(* IEC 61131-3 sources: ConveyorControl-with-PLC/4E_Gruppe1_Graf_Projekt1_HMI/Class/_Lse (part 2) *)

StrChrUniBbB
    LDRB      r3, [p0], #1
    LDRB      r11, [p0], #1
    ORR       r3, r3, r11, LSL #8
    CMP       r3, x1
    BEQ       StrChrEnd
    CMP       r3, #0
    BEQ       StrChrNotFound
    ADD       r10, r10, #1
    B         StrChrUniBbB

StrChrNotFound
    MOV       r10, #65280
    ADD       r10, r10, #255

StrChrEnd
    MOV       retcode, r10
#else //elif _LSL_TARGETARCH_X86
    pushfd
    push      esi

    clr       ebx
    clr       ecx

    l.esi     p0
    o.esi     esi
    jz        StringChrRet

    cld
    l.bx      x1
    cmp.w     x2,1
    jne       StringChrLoopUni

StringChrLoop
    lodsb
    o.al      al
    jz        StringChrRet
    x.al      bl
    jz        StringChrSuccess
    inc       ecx
    jmp       StringChrLoop

StringChrLoopUni
    lodsw
    o.ax      ax
    jz        StringChrRet
    x.ax      bx
    jz        StringChrSuccess
    inc       ecx
    jmp       StringChrLoopUni

StringChrRet
    l.ecx     16#FFFF

StringChrSuccess
    s.cx      retcode

    pop       esi
    popfd
#endif

END_FUNCTION

FUNCTION AWL GLOBAL __CDECL StrXmp
  VAR_INPUT
    pTxt0    : ^void;
    pTxt1    : ^void;
    cSize : UINT;
  END_VAR
  VAR_OUTPUT
    retcode : UDINT;
  END_VAR

#ifdef _LSL_TARGETARCH_ARM
    MOV       retcode, #0

    CMP       pTxt0, pTxt1
    BEQ       StrXmpEnd

    CMP       pTxt0, #0
    BEQ       StrXmpNotEqual
    CMP       pTxt1, #0
    BEQ       StrXmpNotEqual

    CMP       cSize, #1
    BNE       StrXmpUni

StrXmpAscii
    LDRB      r10, [pTxt0], #1
    LDRB      r11, [pTxt1], #1
    CMP       r10, r11
    BNE       StrXmpNotEqual
    CMP       r10, #0
    BEQ       StrXmpEnd
    B         StrXmpAscii

StrXmpUni
    ORR       r11, pTxt0, pTxt1
    TST       r11, #1
    BNE       StrXmpUniBbB   // one or both pointer are missaligned

StrXmpUniH
    LDRH      r10, [pTxt0], #2
    LDRH      r11, [pTxt1], #2
    CMP       r10, r11
    BNE       StrXmpNotEqual
    CMP       r10, #0
    BNE       StrXmpUniH
    B         StrXmpEnd

StrXmpUniBbB
    LDRB      r10, [pTxt0], #1
    LDRB      r3,  [pTxt0], #1
    ORR       r10, r10, r3, LSL #8
    LDRB      r11, [pTxt1], #1
    LDRB      r3,  [pTxt1], #1
    ORR       r11, r11, r3, LSL #8
    CMP       r10, r11
    BNE       StrXmpNotEqual
    CMP       r10, #0
    BNE       StrXmpUniBbB
    B         StrXmpEnd

StrXmpNotEqual
    MOV       retcode, #1

StrXmpEnd

#else //elif _LSL_TARGETARCH_X86
    pushfd
    push      edi
    push      esi

    l.esi     pTxt0
    l.edi     pTxt1
    clr       ecx

    x.esi     edi
    jz        StringXmpEqual

    l.esi     pTxt0
    o.esi     esi
    jz        StringXmpRet
    o.edi     edi
    jz        StringXmpRet

    cld
    cmp.w     cSize,1
    jne       StringXmpLoopUni

StringXmpLoop
    l.cl      (edi)
    or.cl     (esi)
    jecxz     StringXmpEqual
    cmpsb
    jz        StringXmpLoop
    jmp       StringXmpRet

StringXmpLoopUni
    l.cx      (edi)
    or.cx     (esi)
    jecxz     StringXmpEqual
    cmpsw
    jz        StringXmpLoopUni
    //jmp       StringXmpRet

StringXmpRet
    l.ecx     1

StringXmpEqual
    s.ecx     retcode

    pop       esi
    pop       edi

    popfd
#endif

END_FUNCTION

FUNCTION GLOBAL __CDECL get_loaderversion
VAR_OUTPUT
  retcode : UDINT;
END_VAR

  retcode := ops.uiLoaderVersion.usLoRev or (ops.uiLoaderVersion.usHiRev shl 16);

END_FUNCTION

FUNCTION _LookupCls VAR_INPUT pname : ^char; END_VAR VAR_OUTPUT retcode : ^CLSHDR; END_VAR;
FUNCTION GLOBAL __cdecl GetRevisionOfClass VAR_INPUT classname : ^char; END_VAR VAR_OUTPUT retcode : udint; END_VAR
  var
    pClsHdr : ^CLSHDR;
    rhi, rlo : udint;
  end_var

  retcode := 0;
  pClsHdr := _LookupCls(classname);

  if(pClsHdr <> NIL) then
    if(pClsHdr^.pDsc <> NIL) then
      rhi := pClsHdr^.pDsc^.udRev.hi;
      rlo := pClsHdr^.pDsc^.udRev.lo;
      retcode := (rhi shl 16) or rlo;
    end_if;
  end_if;

END_FUNCTION

FUNCTION GLOBAL __CDECL rotate_DOT
VAR_INPUT
  p    : ^_DOT;
  w1   : INT;
END_VAR
VAR
  a1, x, y : _REAL;
  m0, m1 : _REAL;
END_VAR

  x := p^.x;
  y := p^.y;

  a1 := (to_real(w1) * 3.1416) / 180;
  m0 := COS(a1);
  m1 := SIN(a1);

  p^.x := to_int((m0 * x) + (m1 * y));
  p^.y := to_int((m0 * y) - (m1 * x));

END_FUNCTION

FUNCTION GLOBAL __CDECL matrize
VAR_INPUT
  pm : ^_REAL;
  px : ^_REAL;
  py : ^_REAL;
  pz : ^_REAL;
END_VAR
VAR
  x : _REAL;
  y : _REAL;
  z : _REAL;
END_VAR

  x := px^;
  y := py^;
  z := pz^;

  px^ :=( pm^ * x) + ((pm + sizeof(_REAL))^ * y) + ((pm + (sizeof(_REAL) * 2))^ * z);
  py^ := ((pm + (sizeof(_REAL) * 3))^ * x) + ((pm + (sizeof(_REAL) * 4))^ * y) + ((pm + (sizeof(_REAL) * 5))^ * z);
  pz^ := ((pm + (sizeof(_REAL) * 6))^ * x) + ((pm + (sizeof(_REAL) * 7))^ * y) + ((pm + (sizeof(_REAL) * 8))^ * z);

END_FUNCTION

FUNCTION GLOBAL __CDECL rotate_DOT3D
VAR_INPUT
  p    : ^_DOT3D;
  w1   : INT;
  w2   : INT;
  w3   : INT;
END_VAR
VAR
  a1   : _REAL;
  a2   : _REAL;
  a3   : _REAL;
  x    : _REAL;
  y    : _REAL;
  z    : _REAL;
  matr : ARRAY[0..8] of _REAL;
END_VAR

  a1 := w1;
  a2 := w2;
  a3 := w3;

  a1 := (a1 * 3.1416) / 180;
  a2 := (a2 * 3.1416) / 180;
  a3 := (a3 * 3.1416) / 180;

  x := p^.x;
  y := p^.y;
  z := p^.z;

  matr[0] := COS(a1);
  matr[1] := SIN(a1);
  matr[2] := 0;
  matr[3] := -matr[1];
  matr[4] := matr[0];
  matr[5] := 0;
  matr[6] := 0;
  matr[7] := 0;
  matr[8] := 1;
  matrize(#matr[0], #x, #y, #z);

  matr[0] := 1;
  matr[1] := 0;
  matr[2] := 0;
  matr[3] := 0;
  matr[4] := COS(a2);
  matr[5] := SIN(a2);
  matr[6] := 0;
  matr[7] := -matr[5];
  matr[8] := matr[4];
  matrize(#matr[0], #x, #y, #z);

  matr[0] := COS(a3);
  matr[1] := 0;
  matr[2] := SIN(a3);
  matr[3] := 0;
  matr[4] := 1;
  matr[5] := 0;
  matr[6] := -matr[2];
  matr[7] := 0;
  matr[8] := matr[0];
  matrize(#matr[0], #x, #y, #z);

//  p^.x := FTOL(x);
//  p^.y := FTOL(y);
//  p^.z := FTOL(z);

  p^.x := to_int(x);
  p^.y := to_int(y);
  p^.z := to_int(z);

END_FUNCTION

FUNCTION GLOBAL __CDECL AMBDC
VAR_INPUT
  a : UDINT;
  b : UDINT;
  c : UDINT;
END_VAR
VAR_OUTPUT
  retcode : UDINT;
END_VAR

  retcode := a*b/c;

END_FUNCTION

FUNCTION GLOBAL __CDECL heap_size
VAR_INPUT
  total : ^UDINT;
  free  : ^UDINT;
END_VAR
VAR_OUTPUT
  retcode : bool;
END_VAR

  free^  := _UserHeapFreeMem;
  total^ := _UserHeapTotalSize;
  retcode := true;

END_FUNCTION

FUNCTION GLOBAL __CDECL get_microtime
VAR_OUTPUT
  retcode : UDINT;
END_VAR

  retcode := OS_ReadMicroSec();

END_FUNCTION

FUNCTION GLOBAL __CDECL GetResetTaskTime
VAR_INPUT
  pudi : ^UDINT;
END_VAR

  if(pudi <> NIL) then
    pudi^ := _RealMaximumTime;       pudi += 4; // maximum duration of RT-methods
    pudi^ := _RealAverageTime;       pudi += 4; // average duration of RT-methods
    pudi^ := _CyclicMaximumTime;     pudi += 4; // maximum duration of Cy-methods
    pudi^ := _CyclicAverageTime;     pudi += 4; // average duration of Cy-methods
    pudi^ := _BackgroundMaximumTime; pudi += 4; // maximum duration of Bg-methods
    pudi^ := _BackgroundAverageTime;            // average duration of Bg-methods
  else
    _RealMaximumTime       := 0;  // maximum duration of RT-methods
    _RealAverageTime       := 0;  // average duration of RT-methods
    _CyclicMaximumTime     := 0;  // maximum duration of Cy-methods
    _CyclicAverageTime     := 0;  // average duration of Cy-methods
    _BackgroundMaximumTime := 0;  // maximum duration of Bg-methods
    _BackgroundAverageTime := 0;  // average duration of Bg-methods
  end_if;

END_FUNCTION

FUNCTION GLOBAL __CDECL CilGet
VAR_INPUT
	name : ^_ASCII;
	ptr  : ^PVOID;
END_VAR
VAR_OUTPUT
	retcode : BOOL;
END_VAR

  retcode := TRUE;

  if(OS_CILGet(name, ptr) <> SYS_ERR_NONE) then
    ptr^    := NIL;
	retcode := FALSE;
  end_if;

END_FUNCTION

FUNCTION GLOBAL __CDECL GetTCPIPAddressFromDNS
VAR_INPUT
  dnsname   : ^_ASCII;
END_VAR
VAR_OUTPUT
  retcode : UDINT;
END_VAR

  retcode := 0;
  if((lsl_tcp_user <> NIL) & (dnsname <> NIL)) then
    retcode := OS_TCP_USER_STRTOULONG(dnsname);
  end_if;

END_FUNCTION

FUNCTION GLOBAL __CDECL GetTCPIPAddress
VAR_INPUT
  interface : UDINT;
  address   : ^UDINT;
  subnet    : ^UDINT;
  gateway   : ^UDINT;
END_VAR
VAR_OUTPUT
  retcode : BOOL;
END_VAR

  retcode := FALSE;

  if(lsl_tcp_user <> NIL) then
    if(address <> NIL) then
      address^ := 0;
      OS_TCP_USER_IPINFO(interface$DINT, IP_OPT_ADDR, address);
      retcode := TRUE;
    end_if;
    if(subnet <> NIL) then
      subnet^ := 0;
      OS_TCP_USER_IPINFO(interface$DINT, IP_OPT_SUBNETMASK, subnet);
      retcode := TRUE;
    end_if;
    if(gateway <> NIL) then
      gateway^ := 0;
      OS_TCP_USER_IPINFO(interface$DINT, IP_OPT_GATEWAY, gateway);
      retcode := TRUE;
    end_if;
  end_if;

END_FUNCTION

FUNCTION  _Lse::_Lse
VAR_OUTPUT
	ret_code		: CONFSTATES;
END_VAR
VAR
  i : UINT;
  ptr : ^_PICPOI;
END_VAR

  PThis_Lse      := this;
  DownloadState  := 0;
  GlobalBitState := 0;
//LDR_SetWait4Visu(true, 0);

  construct_MAIN();

  mt_api         := NIL;
  Thread2Handle  := NIL;
  MailBox2Handle := NIL;

  if(OS_CILGet("LSL_MULTITASK", #mt_api$void)) THEN
    mt_api := NIL;
  end_if;

  MutexHandler[0] := OS_MT_CreateSemaphore(MTSEMATYPE_MUTEX, 1, 0, "KERNELMUTEX");
  MutexHandler[1] := OS_MT_CreateSemaphore(MTSEMATYPE_MUTEX, 1, 0, "ALARMMUTEX");
  MutexHandler[2] := OS_MT_CreateSemaphore(MTSEMATYPE_MUTEX, 1, 0, "RTK2TASK");
  MutexHandler[3] := OS_MT_CreateSemaphore(MTSEMATYPE_MUTEX, 1, 0, "ReallocREFLIST");
  MutexHandler[4] := OS_MT_CreateSemaphore(MTSEMATYPE_MUTEX, 1, 0, "StartREFLIST");

  OS_pLslSysMsg := NIL;
  if(OS_CILGet("SYSMSG", #OS_pLslSysMsg$void)) THEN
    OS_pLslSysMsg := NIL;
  end_if;

  lsl_tcp_user := NIL;
  if(OS_CILGet("TCP_USER", #lsl_tcp_user$void)) then
    lsl_tcp_user := NIL;
  end_if;

//  init_MAIN();
  init_MEM_POINTERPARA(#UserGlobal);
  init_MEM_POINTER(#Oszis);

  ToolCat    := NIL;
  RunState   := STATE_START;
  ret_code   := C_OK;
  PicMemo.no := 0;
  ptr        := #PicMemo.ptr[0];
  i          := sizeof(PicMemo.ptr) / sizeof(_PICPOI);
  while(i) do
    init_WHOAMI(#ptr^.whoami);
	  ptr^.ptr := NIL;
	  ptr      += sizeof(_PICPOI);
    i        -= 1;
  end_while;

  IsEventProcessor := FALSE;

END_FUNCTION

FUNCTION VIRTUAL GLOBAL _Lse::Init
var
  urinit : bool;
end_var

  if((RunState = STATE_START) | (RunState = STATE_FLY)) then
    urinit := true;
	  if(RunState = STATE_FLY) then
	    urinit := false;
	  end_if;
    RunState := STATE_READY;

    if(RTK_Init(this, urinit) = FALSE) then
	    RunState := STATE_END;
    end_if;
  end_if;

  if(_firstscan) then
    if(IsClientConnected(#EventProcessor) = TRUE) then
      IsEventProcessor := TRUE;
    end_if;

    InitJpgLib();

    if(mt_api <> NIL) then
      if(MailBox2Handle = NIL) then
        MailBox2Handle := OS_MT_CreateMailBox(sizeof(_Thread2CmdLine), 16, "MyMailBox2");
      end_if;

      if(MailBox2Handle <> NIL) & (Thread2Handle = NIL) then
        Thread2Handle := OS_MT_CreateThread(#Thread2(), 9, 8192, 0, this, "MyThread2");
      end_if;
    end_if;
  end_if;

END_FUNCTION

FUNCTION VIRTUAL GLOBAL _Lse::CyWork
VAR_INPUT
EAX		: UDINT;
END_VAR
VAR_OUTPUT
	state		: UDINT;
END_VAR

  state := Background(0);

END_FUNCTION

FUNCTION VIRTUAL GLOBAL _Lse::Background
VAR_INPUT
 EAX  : UDINT;
END_VAR
VAR_OUTPUT
 state  : UDINT;
END_VAR

  if((ops.sysstate = C_RUNRAM) | (ops.sysstate = C_RUNROM)) then

    if(DownloadState = 2) then
      DownloadState := 0;
      new_PLC();
      RTK_End(TRUE);
      RunState := STATE_FLY;
      OfflineMode := 0;
      Init();
    end_if;

    if(RunState = STATE_RUN) then
      if(RTK_Run() = FALSE) then
        if(IF_Stop() = TRUE) then
          MakeLogfile1Entry("End of LSE-task forced by program.", 0, 0);
          RunState := STATE_END;
        end_if;
      end_if;
    elsif(RunState = STATE_READY) then
      RunState   := STATE_RUN;
      if(RTK_Ready() = FALSE) then
        RunState := STATE_END;
      end_if;
    elsif(RunState = STATE_END) then
      RTK_End(FALSE);
      RunState := STATE_ERROR;
    end_if;
  end_if;

  state := READY$UDINT;

END_FUNCTION

FUNCTION __CDECL VIRTUAL GLOBAL _Lse::IF_WindowStart
VAR_INPUT
	whoami		: ^_WHOAMI;
	pic		    : ^VOID;
	firsttime	: BOOL;
END_VAR
VAR
  pp  : ^_PICPOI;
	no  : UDINT;
  ppp : ^_POINTERPARA;
END_VAR

  if(GlobalBitState and GLOBAL_BIT_IFWINSTART) then
    no  := UserGlobal.no;
    ppp := UserGlobal.ptr;
    while no do
      if(ppp^.para and GLOBAL_BIT_IFWINSTART) then
        ppp^.ptr$^_Global^.IF_WindowStart(whoami, pic, firsttime);
      end_if;
	    no  -= 1;
	    ppp += sizeof(_POINTERPARA);
    end_while;
  end_if;

  pp := FindScreen(whoami);
  if(pp <> NIL) then
    pp^.ptr$^_Screen^.S_Start(pic, firsttime);
    pic^$^_Screen := pp^.ptr$^_Screen;
  end_if;

END_FUNCTION

FUNCTION __CDECL VIRTUAL GLOBAL _Lse::IF_WindowReady
VAR_INPUT
	whoami		: ^_WHOAMI;
	pic		    : ^VOID;
	firsttime	: BOOL;
END_VAR
VAR
	no  : UDINT;
	ppp : ^_POINTERPARA;
END_VAR

  if(GlobalBitState and GLOBAL_BIT_IFWINREADY) then
    no  := UserGlobal.no;
    ppp := UserGlobal.ptr;
    while no do
      if(ppp^.para and GLOBAL_BIT_IFWINREADY) then
        ppp^.ptr$^_Global^.IF_WindowReady(whoami, pic, firsttime);
      end_if;
      no  -= 1;
      ppp += sizeof(_POINTERPARA);
    end_while;
  end_if;

  if(pic <> NIL) then
    if(pic^$^_Screen <> NIL) then
      pic^$^_Screen^.S_Ready(pic, firsttime);
    end_if;
  end_if;

END_FUNCTION

FUNCTION __CDECL VIRTUAL GLOBAL _Lse::IF_WindowRun
VAR_INPUT
	whoami		: ^_WHOAMI;
	pic		    : ^VOID;
	event		: ^_EVENT;
END_VAR
VAR
 	no  : UDINT;
	ppp : ^_POINTERPARA;
END_VAR

  if(GlobalBitState and GLOBAL_BIT_IFWINRUN) then
    no  := UserGlobal.no;
    ppp := UserGlobal.ptr;
    while no do
      if(ppp^.para and GLOBAL_BIT_IFWINRUN) then
        ppp^.ptr$^_Global^.IF_WindowRun(whoami, pic, event);
      end_if;
      no  -= 1;
      ppp += sizeof(_POINTERPARA);
    end_while;
  end_if;

  if(pic <> NIL) then
    if(pic^$^_Screen <> NIL) then
      pic^$^_Screen^.S_Run(pic, event);
    end_if;
  end_if;

END_FUNCTION

FUNCTION __CDECL VIRTUAL GLOBAL _Lse::IF_WindowEnd
VAR_INPUT
	whoami		: ^_WHOAMI;
	pic		    : ^VOID;
END_VAR
VAR
  pp  : ^_PICPOI;
	no  : UDINT;
	ppp : ^_POINTERPARA;
END_VAR

  if(GlobalBitState and GLOBAL_BIT_IFWINEND) then
    no  := UserGlobal.no;
    ppp := UserGlobal.ptr;
    while no do
      if(ppp^.para and GLOBAL_BIT_IFWINEND) then
        ppp^.ptr$^_Global^.IF_WindowEnd(whoami, pic);
      end_if;
      no  -= 1;
      ppp += sizeof(_POINTERPARA);
    end_while;
  end_if;

  // parameter 'pic' is used to be NIL therefore use FindScreen
  pp := FindScreen(whoami);
  if(pp <> NIL) then
    pp^.ptr$^_Screen^.S_End(pic);
  end_if;

END_FUNCTION

FUNCTION __CDECL VIRTUAL GLOBAL _Lse::IF_UserCall
VAR_INPUT
	nof	 : DINT;
	para : DINT;
END_VAR
VAR
	no   : UDINT;
	ppp  : ^_POINTERPARA;
END_VAR

  if(GlobalBitState and GLOBAL_BIT_IFUSERCALL) then
    no  := UserGlobal.no;
    ppp := UserGlobal.ptr;
    while no do
      if(ppp^.para and GLOBAL_BIT_IFUSERCALL) then
        ppp^.ptr$^_Global^.IF_UserCall(nof, para);
      end_if;
      no  -= 1;
      ppp += sizeof(_POINTERPARA);
    end_while;
  end_if;

END_FUNCTION

FUNCTION __CDECL VIRTUAL GLOBAL _Lse::IF_AccessInput
VAR_INPUT
	pi		: ^_INPUT;
END_VAR
VAR_OUTPUT
    retcode : BOOL;
END_VAR
VAR
	no   : UDINT;
	ppp  : ^_POINTERPARA;
END_VAR

  retcode := TRUE;

  if(GlobalBitState and GLOBAL_BIT_IFACCESSINPUT) then
    no  := UserGlobal.no;
    ppp := UserGlobal.ptr;
    while no do
      no  -= 1;
      if(ppp^.para and GLOBAL_BIT_IFACCESSINPUT) then
        if(ppp^.ptr$^_Global^.IF_AccessInput(pi) = FALSE) then
          no := 0;
          retcode := FALSE;
        end_if;
      end_if;
      ppp += sizeof(_POINTERPARA);
    end_while;
  end_if;

END_FUNCTION

FUNCTION __CDECL VIRTUAL GLOBAL _Lse::IF_ChkEnable
VAR_INPUT
	key		: DINT;
END_VAR
VAR_OUTPUT
    retcode : BOOL;
END_VAR
VAR
	no   : UDINT;
	ppp  : ^_POINTERPARA;
END_VAR

  retcode := TRUE;

  if(GlobalBitState and GLOBAL_BIT_IFCHKENABLE) then
    no  := UserGlobal.no;
    ppp := UserGlobal.ptr;
    while no do
      no  -= 1;
      if(ppp^.para and GLOBAL_BIT_IFCHKENABLE) then
        if(ppp^.ptr$^_Global^.IF_ChkEnable(key) = FALSE) then
          no := 0;
          retcode := FALSE;
        end_if;
      end_if;
      ppp += sizeof(_POINTERPARA);
    end_while;
  end_if;

END_FUNCTION

FUNCTION __CDECL VIRTUAL GLOBAL _Lse::IF_SystemError
VAR_INPUT
	errno		: DINT;
	para        : DINT;
	ptxt        : ^_CHAR;
END_VAR
VAR_OUTPUT
    retcode : BOOL;
END_VAR
VAR
	no   : UDINT;
	ppp  : ^_POINTERPARA;
END_VAR

  retcode       := TRUE;
  SystemMessage := SystemMessage.Write(errno);

  no  := UserGlobal.no;
  ppp := UserGlobal.ptr;
  while no do
    no  -= 1;
    if(ppp^.ptr$^_Global^.IF_SystemError(errno, para, ptxt) = FALSE) then
      no := 0;
      retcode := FALSE;
    end_if;
    ppp += sizeof(_POINTERPARA);
  end_while;

END_FUNCTION

FUNCTION __CDECL VIRTUAL GLOBAL _Lse::IF_DrawBubbleHelp
VAR_INPUT
	pedit	: ^_EDITOR;
END_VAR
VAR_OUTPUT
    retcode : BOOL;
END_VAR
VAR
	no   : UDINT;
	ppp  : ^_POINTERPARA;
END_VAR

  retcode := TRUE;

  no  := UserGlobal.no;
  ppp := UserGlobal.ptr;
  while no do
    no  -= 1;
    if(ppp^.ptr$^_Global^.IF_DrawBubbleHelp(pedit) = FALSE) then
      no := 0;
      retcode := FALSE;
    end_if;
    ppp += sizeof(_POINTERPARA);
  end_while;

END_FUNCTION

FUNCTION __CDECL VIRTUAL GLOBAL _Lse::IF_UrInit
VAR
	no   : UDINT;
	ppp  : ^_POINTERPARA;
END_VAR

  no  := UserGlobal.no;
  ppp := UserGlobal.ptr;
  while no do
    no  -= 1;
    ppp^.ptr$^_Global^.IF_UrInit();
    ppp += sizeof(_POINTERPARA);
  end_while;

END_FUNCTION

FUNCTION __CDECL VIRTUAL GLOBAL _Lse::IF_ProjectStart
VAR
  no  : UDINT;
  ppp : ^_POINTERPARA;
END_VAR

  no  := UserGlobal.no;
  ppp := UserGlobal.ptr;
  while no do
    no  -= 1;
    ppp^.ptr$^_Global^.IF_ProjectStart();
    ppp += sizeof(_POINTERPARA);
  end_while;

END_FUNCTION

#ifdef UC_MULTICPU
FUNCTION IsSubStationZero
VAR_INPUT
    pcm   : ^_COMAP;
    index : uint;
END_VAR
VAR_OUTPUT
    retcode : BOOL;
END_VAR
VAR
    no : uint;
END_VAR

  retcode := false;
  no      := 256;
  while(no) do
    no -= 1;
    if(pcm^.multimap[0] = index) then
	  retcode := true;
	end_if;
	pcm += sizeof(_COMAP);
  end_while;

END_FUNCTION
#endif

//[#ENGLISH]
//function is called after loading project
//graphic is already initialized,
//no picture is loaded and nothing is on the screen (blank screen)
//state .... TRUE successful loading project, either FALSE
//return FALSE if you don't want to start this application
FUNCTION __CDECL VIRTUAL GLOBAL _Lse::IF_ProjectReady
VAR_INPUT
	state	: BOOL;
END_VAR
VAR_OUTPUT
    retcode : BOOL;
END_VAR
VAR
  no      : UDINT;
	ppp     : ^_POINTERPARA;
  ptrOszi : ^P_Oszi;
  pcs     : ^_COMSET;
  pcp     : ^_COMPORT;
END_VAR

  retcode := state;

  no  := UserGlobal.no;
  ppp := UserGlobal.ptr;
  while no do
    no  -= 1;
    if(ppp^.ptr$^_Global^.IF_ProjectReady(state) = FALSE) then
      no := 0;
      retcode := FALSE;
    end_if;
    ppp += sizeof(_POINTERPARA);
  end_while;

  no := Oszis.no;
  ptrOszi$^UDINT := Oszis.ptr;
  while no do
    no  -= 1;
    if(ptrOszi^^.InitOszi() = FALSE) then
      no := 0;
      retcode := FALSE;
    end_if;
	ptrOszi += 4;
  end_while;

  if(IsClientConnected((#Gbcd)$^DINT) = 1) then
    pcs := Lse_GetComSet();
    no  := pcs^.no;
    pcp := pcs^.ptr;
    while(no) do
      no -= 1;
      if(pcp^.comdef.typ <> _COM_INTERN) then
       #ifdef UC_MULTICPU
        if(IsSubStationZero(#pcs^.mapper[0], to_uint(no)) = true) then
          // geht leider nur von substation 0, alarme sind einfach nur schlecht
          Gbcd.GetLostAlarms(#pcp^.comdef);
        end_if;
       #else
        Gbcd.GetLostAlarms(#pcp^.comdef);
       #endif
      end_if;
	  pcp += sizeof(_COMPORT);
    end_while;
  end_if;

  LseReady := 1;
  if(IsClientConnected((#LseReady)$^DINT) = 1) then
    LseReady.Write(1);
  end_if;

END_FUNCTION

FUNCTION __CDECL VIRTUAL GLOBAL _Lse::IF_ProjectRun
VAR_INPUT
	pe	: ^_EVENT;
END_VAR
VAR
  no  : UDINT;
  ppp : ^_POINTERPARA;
END_VAR

  if(GlobalBitState and GLOBAL_BIT_IFPRJRUN) then
    no  := UserGlobal.no;
    ppp := UserGlobal.ptr;
    while no do
      no  -= 1;
      if(ppp^.para and GLOBAL_BIT_IFPRJRUN) then
        ppp^.ptr$^_Global^.IF_ProjectRun(pe);
      end_if;
      ppp += sizeof(_POINTERPARA);
    end_while;
  end_if;

END_FUNCTION

FUNCTION __CDECL VIRTUAL GLOBAL _Lse::IF_ProjectEnd
VAR
  no  : UDINT;
  ppp : ^_POINTERPARA;
END_VAR

  no  := UserGlobal.no;
  ppp := UserGlobal.ptr;
  while no do
    no  -= 1;
    ppp^.ptr$^_Global^.IF_ProjectEnd();
    ppp += sizeof(_POINTERPARA);
  end_while;

END_FUNCTION

//[#ENGLISH]
//this function is called after a succesfull writing of an input
//pi ......... --> to saved _INPUT
//pr ......... --> to _RESULT
FUNCTION __CDECL VIRTUAL GLOBAL _Lse::IF_InputIsSaved
VAR_INPUT
	pi	: ^_INPUT;
	pr  : ^_RESULT;
END_VAR
VAR
	no   : UDINT;
	ppp  : ^_POINTERPARA;
END_VAR

  no  := UserGlobal.no;
  ppp := UserGlobal.ptr;
  while no do
    no  -= 1;
    ppp^.ptr$^_Global^.IF_InputIsSaved(pi, pr);
    ppp += sizeof(_POINTERPARA);
  end_while;

END_FUNCTION

//[#ENGLISH]
//this method will be called at least (before closing the application).
//note: afterwards there is no more executable code.
FUNCTION __CDECL VIRTUAL GLOBAL _Lse::IF_PowerDown
VAR
	no   : UDINT;
	ppp  : ^_POINTERPARA;
END_VAR

  no  := UserGlobal.no;
  ppp := UserGlobal.ptr;
  while no do
    no  -= 1;
    ppp^.ptr$^_Global^.IF_PowerDown();
    ppp += sizeof(_POINTERPARA);
  end_while;

END_FUNCTION

//[#ENGLISH]
//method is called when input is identified unambiguous by touch and
//the editor can't open because access is denied.
FUNCTION __CDECL VIRTUAL GLOBAL _Lse::IF_InputWithoutAccess
VAR_INPUT
	pi		: ^_INPUT;
	pvi     : ^_VARINFO;
END_VAR
VAR
	no   : UDINT;
	ppp  : ^_POINTERPARA;
END_VAR

  no  := UserGlobal.no;
  ppp := UserGlobal.ptr;
  while no do
    no  -= 1;
    ppp^.ptr$^_Global^.IF_InputWithoutAccess(pi, pvi);
    ppp += sizeof(_POINTERPARA);
  end_while;

END_FUNCTION

//[#ENGLISH]
//method is called when a new alarm is added during runtime to the alarmlist
FUNCTION __CDECL VIRTUAL GLOBAL _Lse::IF_OpenEditor
VAR_INPUT
    pedit : ^_EDITOR;
END_VAR
VAR
	no   : UDINT;
	ppp  : ^_POINTERPARA;
END_VAR

  no  := UserGlobal.no;
  ppp := UserGlobal.ptr;
  while no do
    no  -= 1;
    ppp^.ptr$^_Global^.IF_OpenEditor(pedit);
    ppp += sizeof(_POINTERPARA);
  end_while;

END_FUNCTION

//[#ENGLISH]
//method is called right before data will be written to server
//pres ... --> to data
//pvar ... --> to serverdescription
FUNCTION __CDECL VIRTUAL GLOBAL _Lse::IF_Write
VAR_INPUT
  pres : ^_RESULT;
  pvar : ^_VARIABLE;
END_VAR
VAR_OUTPUT
  retcode : BOOL;
END_VAR
VAR
	no   : UDINT;
	ppp  : ^_POINTERPARA;
END_VAR

  retcode := TRUE;

  no  := UserGlobal.no;
  ppp := UserGlobal.ptr;
  while no do
    no  -= 1;
    if(ppp^.ptr$^_Global^.IF_Write(pres, pvar) = FALSE) then
      no := 0;
      retcode := FALSE;
    end_if;
    ppp += sizeof(_POINTERPARA);
  end_while;

END_FUNCTION

FUNCTION __CDECL VIRTUAL GLOBAL _Lse::IF_CheckPrefix
VAR_INPUT
  varno : UDINT;
  vi    : ^_VARINFO;
END_VAR
VAR_OUTPUT
	retcode		: BOOL;
END_VAR
VAR
	no   : UDINT;
	ppp  : ^_POINTERPARA;
END_VAR

  retcode := FALSE;

  no  := UserGlobal.no;
  ppp := UserGlobal.ptr;
  while no do
    no  -= 1;
    if(ppp^.ptr$^_Global^.IF_CheckPrefix(varno, vi) = TRUE) then
      no := 0;
      retcode := TRUE;
    end_if;
    ppp += sizeof(_POINTERPARA);
  end_while;

END_FUNCTION

FUNCTION __CDECL VIRTUAL GLOBAL _Lse::IF_GetLookUpEmbeddedPointer
VAR_OUTPUT
	retcode		: ^VOID;
END_VAR

  retcode := NIL;

  if((ops.SysState = C_RUNRAM)|(ops.SysState = C_RUNROM)|(ops.SysState = C_OK)) then
    if(_lsl_pos^.piLINKER <> NIL) then
     // if(_lsl_pos^.piLINKER^.LNK_LookupEmbedded <> NIL) then// STR-function from Loader
        retcode := _lsl_pos^.piLINKER^.LNK_LookupEmbedded;
     // end_if;
    end_if;
  end_if;

END_FUNCTION

//[#ENGLISH]
//method is called when a new alarm is added to the alarmlist
FUNCTION GLOBAL _Lse::AddScreen
VAR_INPUT
	ptr		: ^VOID;
	whoami	: ^_WHOAMI;
END_VAR
VAR_OUTPUT
	retcode	: BOOL;
END_VAR
VAR
  pp : ^_PICPOI;
END_VAR

  retcode := TRUE;
  pp      := FindScreen(whoami);

  if(pp <> NIL) then
    pp^.ptr := ptr;
  elsif(PicMemo.no < (sizeof(PicMemo.ptr) / sizeof(_PICPOI))) then
    pp := #PicMemo.ptr[PicMemo.no];
    pp^.whoami := whoami^;
    pp^.ptr    := ptr;
    PicMemo.no += 1;
  else
    retcode    := FALSE;
  end_if;

END_FUNCTION

FUNCTION GLOBAL _Lse::AddGlobal
VAR_INPUT
	ptr		: ^_Global;
END_VAR
VAR_OUTPUT
	retcode		: bool;
END_VAR

  retcode := AddGlobalEx(ptr, 0xFFFFFFFF);

END_FUNCTION

FUNCTION GLOBAL _Lse::AddGlobalEx
VAR_INPUT
	ptr		: ^_Global;
  para : udint;
END_VAR
VAR_OUTPUT
	retcode		: bool;
END_VAR

  retcode := FALSE;
  if(add_MEM_POINTERPARA(#UserGlobal, ptr, para) = TRUE) then
    GlobalBitState := GlobalBitState or para;
    retcode := TRUE;
  end_if;

END_FUNCTION

FUNCTION GLOBAL _Lse::FindScreen
	VAR_INPUT
		whoami 	: ^_WHOAMI;
	END_VAR
	VAR_OUTPUT
		retcode 	: ^_PICPOI;
	END_VAR
VAR
  no : UINT;
  pp : ^_PICPOI;
END_VAR

  retcode := NIL;
  if(PicMemo.no > 0) then
    no := PicMemo.no;
    pp := #PicMemo.ptr[0];
    while no do
      no -= 1;
      if(pp^.whoami.no = whoami^.no) then
        if((pp^.whoami.ima = whoami^.ima) | ((whoami^.ima = IMA_TOUCHEDITOR) & (pp^.whoami.ima = IMA_WINDOW))) then
          retcode  := pp;
          return;
        end_if;
      end_if;
      pp += sizeof(_PICPOI);
    end_while;
  end_if;

END_FUNCTION

FUNCTION GLOBAL _Lse::GetReady
VAR_OUTPUT
	retcode		: BOOL;
END_VAR

  retcode := FALSE;
  if(RunState = STATE_RUN) then
    retcode := TRUE;
  end_if;

END_FUNCTION

//[#ENGLISH]
//this method is called by the kernel to set statusserver like 'language' etc.
//the first parameter is used as schedular which server is to initialize with value (second parameter)
FUNCTION __CDECL VIRTUAL GLOBAL _Lse::IF_SetStatus
VAR_INPUT
  no    : DINT;
  value : DINT;
END_VAR

// no - Which server has to be changed
// 0...language
// 1...compiler-version
// 2...lse-version
// 3...delaytime screensaver
// 4...commasign
// 5...american date format
// 6...seek algorithm

  case no of
    LSE_COMPILERVERSION      : CompilerVersion    := value;
    LSE_LSEVERSION           : LseVersion         := value;
    LSE_LANGUAGE             : Language           := value;
    LSE_SCREENDELAY	         : DelayScreenSaver   := to_udint(value);
    LSE_DIRECTIONONENTER     : DirectionOnEnter   := value;
    LSE_OFFLINEMODE          : OfflineMode        := value;
    LSE_OPSYSVERSION         : OpSysVersion.Read();
    LSE_COMMASIGN            : Commasign.Write(value);
    LSE_AMERICANDATEFORMAT   : AmericanDateFormat.Write(value);
    LSE_AMERICANTIMEFORMAT   : AmericanTimeFormat.Write(value);
    LSE_SEEKALGORITHM        : SeekAlgorithm.Write(value);
    LSE_CURSORWRAPHORIZONTAL : CursorWrapHorizontal.Write(value);
    LSE_CURSORWRAPVERTICAL   : CursorWrapVertical.Write(value);
    LSE_NOEXTERNCOM          : NoExternCom.Write(value);
    LSE_ACTIVATEBUBBLEHELP   : ActivateBubbleHelp := value;
    LSE_LSEREVISION          : LseProjectRevision := value$hdint;
  end_case;

END_FUNCTION

FUNCTION __CDECL VIRTUAL GLOBAL _Lse::IF_GetStatus
VAR_INPUT
	no		: DINT;
END_VAR
VAR_OUTPUT
	retcode		: DINT;
END_VAR

  case no of
    LSE_LANGUAGE             : retcode := Language;
    LSE_SCREENDELAY	         : retcode$UDINT := DelayScreenSaver;
    LSE_DIRECTIONONENTER     : retcode := DirectionOnEnter;
    LSE_COMMASIGN            : retcode := Commasign;
    LSE_AMERICANDATEFORMAT   : retcode := AmericanDateFormat;
    LSE_AMERICANTIMEFORMAT   : retcode := AmericanTimeFormat;
    LSE_SEEKALGORITHM        : retcode := SeekAlgorithm;
    LSE_CURSORWRAPHORIZONTAL : retcode := CursorWrapHorizontal;
    LSE_CURSORWRAPVERTICAL   : retcode := CursorWrapVertical;
    LSE_LSEVERSION           : retcode := LseVersion;
    LSE_NOEXTERNCOM          : retcode := NoExternCom;
    LSE_ACTIVATEBUBBLEHELP   : retcode := ActivateBubbleHelp;
    LSE_LSEREVISION          : retcode$HDINT := LseProjectRevision;
  end_case;

END_FUNCTION

FUNCTION __CDECL VIRTUAL GLOBAL _Lse::IF_Trace
VAR_INPUT
	msg		: ^_ASCII;
END_VAR

  Trace(msg);

END_FUNCTION

FUNCTION __CDECL VIRTUAL GLOBAL _Lse::IF_GetHeapInfo
VAR_INPUT
	pr : ^_ROOM;
END_VAR

  draw_heap(pr);

END_FUNCTION

FUNCTION __CDECL VIRTUAL GLOBAL _Lse::IF_FoundSomethingByHid
VAR_INPUT
	ima		: _FOUNDHID;
END_VAR
VAR
	no  : UDINT;
	ppp  : ^_POINTERPARA;
END_VAR

  if(GlobalBitState and GLOBAL_BIT_IFFOUNDHID) then
    no  := UserGlobal.no;
    ppp := UserGlobal.ptr;
    while no do
      if(ppp^.para and GLOBAL_BIT_IFFOUNDHID) then
        ppp^.ptr$^_Global^.IF_FoundSomethingByHid(ima);
      end_if;
      no  -= 1;
      ppp += sizeof(_POINTERPARA);
    end_while;
  end_if;

END_FUNCTION

//[#ENGLISH]
//method is called by the kernel right before a menu will be opend.
//the first parameter is a pointer to structure where the menudata like color,
//shape, lines etc. will be stored
//the second parameter is a pointer to the menunumber initialiced by lse
FUNCTION __CDECL VIRTUAL GLOBAL _Lse::IF_PopUpCall
VAR_INPUT
	pm		: ^_MENU;
	pno		: ^UINT;
END_VAR
VAR_OUTPUT
	retcode		: BOOL;
END_VAR
VAR
	no  : UDINT;
	ppp  : ^_POINTERPARA;
END_VAR

  retcode := FALSE;

  no  := UserGlobal.no;
  ppp := UserGlobal.ptr;
  while no do
    no  -= 1;
    if(ppp^.ptr$^_Global^.IF_PopUpCall(pm, pno) = TRUE) then
      retcode := TRUE;
      no := 0;
    end_if;
    ppp += sizeof(_POINTERPARA);
  end_while;

END_FUNCTION

FUNCTION GLOBAL _Lse::AddOszi
VAR_INPUT
	ptr		: ^_OsziLSE;
END_VAR
VAR_OUTPUT
	retcode		: bool;
END_VAR

  retcode := FALSE;
  if(add_MEM_POINTER(#Oszis, ptr) = TRUE) then
    retcode := TRUE;
  end_if;

END_FUNCTION

FUNCTION __CDECL VIRTUAL GLOBAL _Lse::IF_OpenTouchEditor
VAR_INPUT
	pe        : ^_EDITOR;
	preselect : UINT;
END_VAR
VAR_OUTPUT
	retcode		: UINT;
END_VAR
VAR
	no  : UDINT;
	ppp  : ^_POINTERPARA;
END_VAR

  retcode := preselect;

  no  := UserGlobal.no;
  ppp := UserGlobal.ptr;
  while no do
    no  -= 1;
    retcode := ppp^.ptr$^_Global^.IF_OpenTouchEditor(pe, preselect);
    if(retcode <> preselect) then
      no := 0;
    end_if;
    ppp += sizeof(_POINTERPARA);
  end_while;

END_FUNCTION

FUNCTION __CDECL VIRTUAL GLOBAL _Lse::IF_AccessButton
VAR_INPUT
  pb        : ^_BUTTON;
END_VAR
VAR_OUTPUT
  retcode		: BOOL;
END_VAR
VAR
	no   : UDINT;
	ppp  : ^_POINTERPARA;
END_VAR

  retcode := TRUE;

  if(GlobalBitState and GLOBAL_BIT_IFACCESSBUTTON) then
    no  := UserGlobal.no;
    ppp := UserGlobal.ptr;
    while no do
      no -= 1;
      if(ppp^.para and GLOBAL_BIT_IFACCESSBUTTON) then
        if(ppp^.ptr$^_Global^.IF_AccessButton(pb) = FALSE) then
          no := 0;
          retcode := FALSE;
        end_if;
      end_if;
      ppp += sizeof(_POINTERPARA);
    end_while;
  end_if;

END_FUNCTION

FUNCTION GLOBAL _Lse::SetThisPointer
VAR_INPUT
	pointer		: ^void;
	index		: UINT;
END_VAR

  case index of
    0 : ToolCat := pointer;
  end_case;

END_FUNCTION

FUNCTION __CDECL VIRTUAL GLOBAL _Lse::IF_GetThisPointer
VAR_INPUT
	index		: UINT;
END_VAR
VAR_OUTPUT
	retcode		: ^void;
END_VAR

  retcode := NIL;

  case index of
    0 : retcode := ToolCat;
  end_case;

END_FUNCTION

FUNCTION VIRTUAL GLOBAL _Lse::Language::Write
VAR_INPUT
	input		: DINT;
END_VAR
VAR_OUTPUT
	result		: DINT;
END_VAR

  InsertCmd(CMD_NEWLANGUAGE, input, 0);
  result := 1;

END_FUNCTION

FUNCTION VIRTUAL GLOBAL _Lse::DelayScreenSaver::Write
	VAR_INPUT
		input (EAX) 	: UDINT;
	END_VAR
	VAR_OUTPUT
		result (EAX) 	: UDINT;
	END_VAR

	DelayScreenSaver := input$UDINT;
    set_delay_screensave(input$UDINT);
	result := 1;

END_FUNCTION

FUNCTION VIRTUAL GLOBAL _Lse::DelayScreenSaver::Read
	VAR_OUTPUT
		output (EAX) 	: UDINT;
	END_VAR

    DelayScreenSaver := get_delay_screensave();
    output := DelayScreenSaver;

END_FUNCTION

FUNCTION VIRTUAL GLOBAL _Lse::CommaSign::Write
VAR_INPUT
	input		: DINT;
END_VAR
VAR_OUTPUT
	result		: DINT;
END_VAR
VAR
    tmp : BOOL;
END_VAR

  tmp := FALSE;
  if(input) then
    tmp := TRUE;
  end_if;

  CommaSign := tmp;
  set_commasign(tmp);
  result := 1;

END_FUNCTION

FUNCTION VIRTUAL GLOBAL _Lse::CommaSign::Read
VAR_OUTPUT
	output		: DINT;
END_VAR

  CommaSign := get_commasign();
  output := TO_DINT(CommaSign);

END_FUNCTION

FUNCTION VIRTUAL GLOBAL _Lse::AmericanDateFormat::Write
VAR_INPUT
	input		: DINT;
END_VAR
VAR_OUTPUT
	result		: DINT;
END_VAR
VAR
    tmp : BOOL;
END_VAR

  tmp := FALSE;
  if(input) then
    tmp := TRUE;
  end_if;

  AmericanDateFormat := tmp;
  set_americandateformat(tmp);
  result := 1;

END_FUNCTION

FUNCTION VIRTUAL GLOBAL _Lse::AmericanDateFormat::Read
VAR_OUTPUT
	output		: DINT;
END_VAR

  AmericanDateFormat := get_americandateformat();
  output := TO_DINT(AmericanDateFormat);

END_FUNCTION

FUNCTION VIRTUAL GLOBAL _Lse::AmericanTimeFormat::Write
VAR_INPUT
	input		: DINT;
END_VAR
VAR_OUTPUT
	result		: DINT;
END_VAR
VAR
    tmp : BOOL;
END_VAR

  tmp := FALSE;
  if(input) then
    tmp := TRUE;
  end_if;

  AmericanTimeFormat := tmp;
  set_americantimeformat(tmp);
  result := 1;

END_FUNCTION

FUNCTION VIRTUAL GLOBAL _Lse::AmericanTimeFormat::Read
VAR_OUTPUT
	output		: DINT;
END_VAR

  AmericanTimeFormat := get_americantimeformat();
  output := TO_DINT(AmericanTimeFormat);

END_FUNCTION

FUNCTION VIRTUAL GLOBAL _Lse::GotAlarm::Write
VAR_INPUT
	input		: DINT;
END_VAR
VAR_OUTPUT
	result		: DINT;
END_VAR
VAR
  pac : ^_ALACELL;
  check : BOOL;
END_VAR

  result := input;
  check  := TRUE;
  pac    := input$^_ALACELL;

  if(pac^.kennung and 2#00000010) then
    pac^.kennung := pac^.kennung and 2#11111101;  // GetLostAlarms Kennung entfernen
    check := CheckLostAlarm(pac);
 #ifdef USER_BILLION
  elsif (LseReady = 0) & (IsClientConnected((#Gbcd)$^DINT) = 1) then
    if Gbcd.Server0.read() then
      check := FALSE; // RamAnd 2007-04-27 Bei Mehrprozessorlösungen keine Alarme annehmen (von verbundenem Gbcd),
    end_if;           // bevor Lse bereit ist (sonst Alarme doppelt in Liste)
 #endif
  end_if;

  if(check = TRUE) then
    store_ALACELL(pac);
  end_if;

  GotAlarm := input;

END_FUNCTION

FUNCTION VIRTUAL GLOBAL _Lse::SeekAlgorithm::Read
VAR_OUTPUT
	output		: DINT;
END_VAR

  if(get_seek_algorithm() = FALSE) then
    output :=
	SeekAlgorithm := 0;
  else
    output :=
	SeekAlgorithm := 1;
  end_if;

END_FUNCTION

FUNCTION VIRTUAL GLOBAL _Lse::SeekAlgorithm::Write
VAR_INPUT
	input		: DINT;
END_VAR
VAR_OUTPUT
	result		: DINT;
END_VAR
VAR
    tmp : BOOL;
END_VAR

  tmp := FALSE;
  if(input) then
    tmp := TRUE;
  end_if;

  set_seek_algorithm(tmp);
  SeekAlgorithm := tmp;
  result := 1;

END_FUNCTION

FUNCTION VIRTUAL GLOBAL _Lse::OpSysVersion::Read
	VAR_OUTPUT
		output (EAX) 	: UDINT;
	END_VAR

  OpSysVersion := _RTOSVERSION;
  output := OpSysVersion;

END_FUNCTION

FUNCTION VIRTUAL GLOBAL _Lse::DirectionOnEnter::Write
VAR_INPUT
	input		: DINT;
END_VAR
VAR_OUTPUT
	result		: DINT;
END_VAR
VAR
    tmp : BOOL;
END_VAR

  tmp := FALSE;
  if(input) then
    tmp := TRUE;
  end_if;

  DirectionOnEnter := tmp;
  set_directiononenter(tmp);
  result := 1;

END_FUNCTION

FUNCTION VIRTUAL GLOBAL _Lse::CursorWrapHorizontal::Write
VAR_INPUT
	input		: DINT;
END_VAR
VAR_OUTPUT
	result		: DINT;
END_VAR
VAR
    tmp : BOOL;
END_VAR

  tmp := FALSE;
  if(input) then
    tmp := TRUE;
  end_if;

  CursorWrapHorizontal := tmp;
  set_cursorwraphorizontal(tmp);
  result := 1;

END_FUNCTION

FUNCTION VIRTUAL GLOBAL _Lse::CursorWrapVertical::Write
VAR_INPUT
	input		: DINT;
END_VAR
VAR_OUTPUT
	result		: DINT;
END_VAR
VAR
    tmp : BOOL;
END_VAR

  tmp := FALSE;
  if(input) then
    tmp := TRUE;
  end_if;

  CursorWrapVertical := tmp;
  set_cursorwrapvertical(tmp);
  result := 1;

END_FUNCTION

FUNCTION VIRTUAL GLOBAL _Lse::OfflineMode::Write
VAR_INPUT
	input		: DINT;
END_VAR
VAR_OUTPUT
	result		: DINT;
END_VAR

  result := ACCESS_DENIED;
  if(input = 0) then
    if(OfflineMode <> 0) then
	  result := 0;
      InsertCmd(CMD_RECONFIGVAR, 0, 0);
	  end_if;
  end_if;

END_FUNCTION

FUNCTION VIRTUAL GLOBAL _Lse::NoExternCom::Write
VAR_INPUT
	input		: DINT;
END_VAR
VAR_OUTPUT
	result		: DINT;
END_VAR
VAR
    tmp : BOOL;
END_VAR

  tmp := FALSE;
  if(input) then
    tmp := TRUE;
  end_if;

  NoExternCom := tmp;
  set_noexterncom(tmp);
  result := 1;

END_FUNCTION

//[#ENGLISH]
//Interface is called right after language has changed
//parameter actno is number of actual language
//parameter oldno is number of previous language
FUNCTION __CDECL VIRTUAL GLOBAL _Lse::IF_LanguageHasChanged
VAR_INPUT
	actno		: UINT;
	oldno		: UINT;
END_VAR
VAR
	no  : UDINT;
	ppp  : ^_POINTERPARA;
END_VAR

  no  := UserGlobal.no;
  ppp := UserGlobal.ptr;
  while no do
    ppp^.ptr$^_Global^.IF_LanguageHasChanged(actno, oldno);
    no  -= 1;
    ppp += sizeof(_POINTERPARA);
  end_while;

END_FUNCTION

FUNCTION __CDECL VIRTUAL GLOBAL _Lse::IF_LanguageWillChange
VAR_INPUT
	newno		: UINT;
	oldno		: UINT;
END_VAR
VAR
	no  : UDINT;
	ppp  : ^_POINTERPARA;
END_VAR

  no  := UserGlobal.no;
  ppp := UserGlobal.ptr;
  while no do
    ppp^.ptr$^_Global^.IF_LanguageWillChange(newno, oldno);
    no  -= 1;
    ppp += sizeof(_POINTERPARA);
  end_while;

END_FUNCTION

FUNCTION __CDECL VIRTUAL GLOBAL _Lse::IF_Offline
VAR_INPUT
	station		: UINT;
END_VAR
VAR
	no   : UDINT;
	ppp  : ^_POINTERPARA;
END_VAR

  no  := UserGlobal.no;
  ppp := UserGlobal.ptr;
  while no do
    ppp^.ptr$^_Global^.IF_Offline(station);
    no  -= 1;
    ppp += sizeof(_POINTERPARA);
  end_while;

END_FUNCTION

FUNCTION __CDECL VIRTUAL GLOBAL _Lse::IF_OverloadEditor
VAR_INPUT
    pm          : ^_PICTUREMASK;
	whoami		: ^_WHOAMI;
	pvl		: ^_VARLABEL;
END_VAR
VAR
	no   : UDINT;
	ppp  : ^_POINTERPARA;
END_VAR

  no  := UserGlobal.no;
  ppp := UserGlobal.ptr;
  while no do
    ppp^.ptr$^_Global^.IF_OverloadEditor(pm, whoami, pvl);
    no  -= 1;
    ppp += sizeof(_POINTERPARA);
  end_while;

END_FUNCTION

FUNCTION __CDECL VIRTUAL GLOBAL _Lse::IF_ConfigDriveList
VAR_INPUT
	drvlst		: ^char;
	pthis		: ^void;
END_VAR
VAR
	no   : UDINT;
	ppp  : ^_POINTERPARA;
END_VAR

  no  := UserGlobal.no;
  ppp := UserGlobal.ptr;
  while no do
    ppp^.ptr$^_Global^.IF_ConfigDriveList(drvlst, pthis);
    no  -= 1;
    ppp += sizeof(_POINTERPARA);
  end_while;

END_FUNCTION

#ifndef UC_IPC
FUNCTION GLOBAL __CDECL RealComp
VAR_INPUT
  a : ^REAL;
  b : ^REAL;
  op : UINT;
END_VAR
VAR_OUTPUT
  retcode : _BOOL;
END_VAR

  retcode := _FALSE;

  case op of
    IOP_OR:            // logic ||
      if(a^ | b^) then
        retcode := _TRUE;
      end_if;
    IOP_AND:           // logic &&
      if(a^ & b^) then
        retcode := _TRUE;
      end_if;
    IOP_SMALLER:       // logic <
      if(a^ < b^) then
        retcode := _TRUE;
      end_if;
    IOP_SMALLEREQUAL:  // logic <=
      if(a^ <= b^) then
        retcode := _TRUE;
      end_if;
    IOP_EQUAL:         // logic ==
      if(a^ = b^) then
        retcode := _TRUE;
      end_if;
    IOP_BIGGER:        // logic >
      if(a^ > b^) then
        retcode := _TRUE;
      end_if;
    IOP_BIGGEREQUAL:   // logic >=
      if(a^ >= b^) then
        retcode := _TRUE;
      end_if;

  end_case;

END_FUNCTION

FUNCTION GLOBAL __CDECL RealCalc
VAR_INPUT
  ret : ^_REAL;
  a : ^REAL;
  b : ^REAL;
  op : UINT;
END_VAR

  case op of
    IOP_A_PLUS:        // arithmetic +
      ret^ := a^ + b^;
    IOP_A_MINUS:       // arithmetic -
      ret^ := a^ - b^;
    IOP_A_MULTI:       // arithmetic *
      ret^ := a^ * b^;
    IOP_A_DIV:         // arithmetic /
      ret^ := a^ / b^;
    IOP_A_MOD:         // arithmetic %
      ret^ := a^ mod b^;
    IOP_A_OR:          // arithmetic |
      ret^ := a^ or b^;
    IOP_A_AND:         // arithmetic &
      ret^ := a^ and b^;
    IOP_A_EQUAL:       // arithmetic =
      ret^ := a^;

  end_case;

END_FUNCTION

FUNCTION GLOBAL __CDECL ftol_
VAR_INPUT
  a : ^_REAL;
END_VAR
VAR_OUTPUT
  ret : _DWORD;
END_VAR

  ret := to_dint(a^);

END_FUNCTION

FUNCTION GLOBAL __CDECL format_value_st
VAR_INPUT
	value : ^REAL;
	pi    : ^_VARINFO;
  dezpt : _UWORD;
END_VAR
VAR_OUTPUT
  retcode : _IVALUE;
END_VAR
VAR
  tempr : _REAL;
END_VAR

  retcode$REAL := value^;

  if((pi^.vartype = BINARY) & (pi^.format = SIZE_REAL)) then

    tempr := value^;

    if(tempr >= 0) then
      retcode := to_dint((tempr * to_real(get_multiplicator(dezpt))) + 0.5);
    else
      retcode := to_dint((tempr * to_real(get_multiplicator(dezpt))) - 0.5);
    end_if;

  end_if;

END_FUNCTION

FUNCTION GLOBAL __CDECL RealToStr
VAR_INPUT
  txt : ^void;
  value : _REAL;
  dzp : UINT;
  chr_size : UINT;
END_VAR
VAR
  vk  : DINT;
  nk  : DINT;
  len : UINT;
END_VAR
  // dzp ... anzahl der gültigen nachkommastellen

  vk := TO_DINT(value);
  DToA(txt, vk, 0x0800, chr_size);

  if(dzp <> 0) then
    nk  := TO_DINT((value - TO_REAL(vk)) * TO_REAL(get_multiplicator(dzp)));
    len := StrLen(txt, chr_size);
	StrCat(txt, chr_size, ".", sizeof(_ASCII));
    txt += (len + 1) * chr_size;
    DToA(txt, nk, 0x0800, chr_size);
  end_if;

END_FUNCTION

FUNCTION GLOBAL __CDECL StrToReal
VAR_INPUT
  dv : ^_REAL;
  txt : ^void;
  chr_size : _UWORD;
END_VAR
VAR_OUTPUT
  retcode : _BOOL;
END_VAR
VAR
  neg : _BOOL;
  dot : _BOOL;
  run : _BOOL;
  vk : _DWORD;
  nk : _DWORD;
  div : _UWORD;
  rval : _REAL;
  atx : ^_ASCII;
  ac : _ASCII;
END_VAR

  retcode := _FALSE;
  neg := _FALSE;
  dot := _FALSE;
  run := _TRUE;
  vk := 0;
  nk := 0;
  div := 1;
  rval := 0;

  if(chr_size = 1) then
    atx := txt$^_ASCII;
    repeat
      ac := atx^;
      if(ac = '-') then
        neg := _TRUE;
      elsif((ac = '.')|(ac = ',')) then
        dot := _TRUE;
      elsif((ac >= '0') & (ac <= '9')) then
        retcode := _TRUE;
        if(dot = _FALSE) then
          vk := (vk * 10) + (ac - '0');
        else
          div := div * 10;
          nk := (nk * 10) + (ac - '0');
        end_if;
      elsif(ac = 0) then
        run := _FALSE;
      end_if;

      atx += 1;

		until(run = _FALSE)
    end_repeat;

  end_if;

  if(retcode = _TRUE) then
    rval := vk;

    if((div > 1) & (nk <> 0)) then
      rval := rval + ((to_real(nk)) / div);
    end_if;
  end_if;

  if(neg = _TRUE) then
    rval := -rval;
  end_if;

  dv^ := rval;

END_FUNCTION

FUNCTION GLOBAL __CDECL string_to_value
VAR_INPUT
  x0 : DINT;
  p1 : ^_VARINFO;
END_VAR
VAR_OUTPUT
  retcode : DINT;
END_VAR

  retcode := x0;

 #ifdef UC_REAL
  if((p1^.vartype = BINARY) & (p1^.format = SIZE_REAL)) then
    retcode$REAL := ((to_real(x0) / TO_REAL(get_multiplicator(TO_UINT(VarList_GetDezPoint(p1))))));
  end_if;
 #endif

END_FUNCTION

FUNCTION GLOBAL __CDECL MakeMinMax
VAR_INPUT
  dz   : ^_RESULT;
  sz   : ^_RESULT;
  minz : BOOL;
END_VAR
VAR
  rval : REAL;
  dval : DINT;
END_VAR

 #ifdef UC_REAL
  if(dz^.ftype = RES_REAL) then
    if((sz^.ftype = RES_CONSTANT)|(sz^.ftype = RES_NUMERIC)) then
      rval := TO_REAL(sz^.value);
    elsif(sz^.ftype = RES_REAL) then
      rval := sz^.value$REAL;
    end_if;

    if(minz = _TRUE) then

      if(rval > dz^.rmin$REAL) then
        dz^.rmin$REAL := rval;
      end_if;
    else
      if(rval < dz^.rmax$REAL) then
        dz^.rmax$REAL := rval;
      end_if;
    end_if;

    return;

  end_if;
 #endif

  if((sz^.ftype = RES_CONSTANT)|(sz^.ftype = RES_NUMERIC)) then
    dval := sz^.value;
  else
    dval := TO_DINT(sz^.value$REAL);
  end_if;

  if(minz = _TRUE) then
    if(dval > dz^.rmin) then
      dz^.rmin := dval;
    end_if;
  else
    if(dval < dz^.rmax) then
      dz^.rmax := dval;
    end_if;
  end_if;

END_FUNCTION

FUNCTION GLOBAL __CDECL dword2real
VAR_INPUT
  a : ^_REAL;
  b : _DWORD;
END_VAR

  a^ := to_real(b);

END_FUNCTION

#endif

FUNCTION GetMulDiv VAR_INPUT einheit:UDINT; posdezpt:DINT; END_VAR VAR_OUTPUT retcode:UDINT; END_VAR
  var
    dekade : dint;
  end_var

  dekade := 0;
  case(einheit) of
    1000000000 : dekade := 9;
    100000000  : dekade := 8;
    10000000   : dekade := 7;
    1000000    : dekade := 6;
    100000     : dekade := 5;
    10000      : dekade := 4;
    1000       : dekade := 3;
    100        : dekade := 2;
    10         : dekade := 1;
  end_case;

  retcode := 1;
  case(dekade - posdezpt) of
    9 : retcode := 1000000000;
    8 : retcode :=  100000000;
    7 : retcode :=   10000000;
    6 : retcode :=    1000000;
    5 : retcode :=     100000;
    4 : retcode :=      10000;
    3 : retcode :=       1000;
    2 : retcode :=        100;
    1 : retcode :=         10;
  end_case;

END_FUNCTION

FUNCTION MyRealCalc VAR_INPUT value:REAL; posdezpt:DINT; direction:BOOL; END_VAR VAR_OUTPUT retcode:REAL; END_VAR
  var
    div : REAL;
  end_var

  div := 1.0;
  case(posdezpt) of
    1 : div :=     10.0;
    2 : div :=    100.0;
    3 : div :=   1000.0;
    4 : div :=  10000.0;
  end_case;

  if(direction = true) then
    if(value < 0) then
      retcode := ((value * div) - 0.5);
	else
      retcode := ((value * div) + 0.5);
    end_if;
  else
    if(value < 0) then
      retcode := ((value / div) - 0.5);
    else
      retcode := ((value / div) + 0.5);
    end_if;
  end_if;

END_FUNCTION

FUNCTION R_Stroke2mm VAR_INPUT v:REAL; p:^_VARIABLE; d:BOOL; END_VAR VAR_OUTPUT r:REAL; END_VAR

  if(d = true) then // stroke -> mm
    r := v  / (1mm);
  else // mm -> stroke
    r := v * (1mm);
  end_if;

END_FUNCTION

FUNCTION R_Temp2Celsius VAR_INPUT v:REAL; p:^_VARIABLE; d:BOOL; END_VAR VAR_OUTPUT r:REAL; END_VAR

  if(d = true) then
    r := v / 10.0;
  else
    r := v * 10.0;
  end_if;

END_FUNCTION

FUNCTION R_Weight2Kilogram VAR_INPUT v:REAL; p:^_VARIABLE; d:BOOL; END_VAR VAR_OUTPUT r:REAL; END_VAR

  if(d = true) then
    r := v / 10000.0;
  else
    r := v * 10000.0;
  end_if;

END_FUNCTION

FUNCTION R_Time2Second VAR_INPUT v:REAL; p:^_VARIABLE; d:BOOL; END_VAR VAR_OUTPUT r:REAL; END_VAR

  if(d = true) then
    r := v / (1.0sec);
  else
    r := v * (1.0sec);
  end_if;

END_FUNCTION

FUNCTION R_Time2Minute VAR_INPUT v:REAL; p:^_VARIABLE; d:BOOL; END_VAR VAR_OUTPUT r:REAL; END_VAR

  if(d = true) then
    r := R_Time2Second((v + 30)/60, p, true);
  else
    r := R_Time2Second(v*60, p, false);
  end_if;

END_FUNCTION

FUNCTION R_Time2Hour VAR_INPUT v:REAL; p:^_VARIABLE; d:BOOL; END_VAR VAR_OUTPUT r:REAL; END_VAR

  if(d = true) then
    r := R_Time2Minute((v + 30)/60, p, true);
  else
    r := R_Time2Minute(v*60, p, false);
  end_if;

END_FUNCTION

FUNCTION R_Pressure2Bar VAR_INPUT v:REAL; p:^_VARIABLE; d:BOOL; END_VAR VAR_OUTPUT r:REAL; END_VAR

  if(d = true) then
    r := v / (1bar); // pressure -> bar
  else
    r := v * (1bar); // bar -> pressure
  end_if;

END_FUNCTION

FUNCTION R_Stroke2inch VAR_INPUT v:REAL; p:^_VARIABLE; d:BOOL; END_VAR VAR_OUTPUT r:REAL; END_VAR

  if(d = true) then // stroke -> inch
    r := v / (25.4mm);
  else  // inch -> stroke
    r := v * (25.4mm);
  end_if;

END_FUNCTION

FUNCTION R_Pressure2Psi VAR_INPUT v:REAL; p:^_VARIABLE; d:BOOL; END_VAR VAR_OUTPUT r:REAL; END_VAR

  // 1bar = 14.50376808 psi
  if(d = true) then // pressure -> psi
    r := (v * (14.50376808)) / (1.0 bar);
  else // psi -> pressure
    r := (v * (1.0bar)) / (14.50376808);
  end_if;

END_FUNCTION

FUNCTION R_Weight2Pound VAR_INPUT v:REAL; p:^_VARIABLE; d:BOOL; END_VAR VAR_OUTPUT r:REAL; END_VAR

  if(d = true) then
    r := (v * 2.205) / 10000.0;
  else
    r := (v * 10000.0) /  2.205;
  end_if;

END_FUNCTION

FUNCTION R_Temp2Fahrenheit VAR_INPUT v:REAL; p:^_VARIABLE; d:BOOL; END_VAR VAR_OUTPUT r:REAL; END_VAR
  // lasal grundeinheit : 10E-1 Grad C
  // [C] = ([F]-32)*5/9

  if(d = true) then
    r := 32.0 + (v * 9.0) / 50.0;
  else
    r := ((v - 32.0) * 50.0) / 9.0;
  end_if;

END_FUNCTION

FUNCTION R_Force2KN VAR_INPUT v:REAL; p:^_VARIABLE; d:BOOL; END_VAR VAR_OUTPUT r:REAL; END_VAR

  if(d = true) then
    r := v  / (1.0 kn); // stroke -> mm
  else
    r := v * (1.0 kn); // mm -> stroke
  end_if;

END_FUNCTION

FUNCTION S_Stroke2mm VAR_INPUT v:DINT; p:^_VARIABLE; d:BOOL; END_VAR VAR_OUTPUT r:DINT; END_VAR

  r$udint := GetMulDiv(1mm, p^.info.posdezpt);

  if(d = true) then // stroke -> mm
    if(v < 0) then
      r := (v - (r/2)) / r;
	else
      r := (v + (r/2)) / r;
    end_if;
  else // mm -> stroke
    r := v * r;
  end_if;

END_FUNCTION

FUNCTION S_Temp2Celsius VAR_INPUT v:DINT; p:^_VARIABLE; d:BOOL; END_VAR VAR_OUTPUT r:DINT; END_VAR

  r$udint := GetMulDiv(10, p^.info.posdezpt);

  if(d = true) then // temperature -> C
    if(v < 0) then
      r := (v - (r/2)) / r;
	else
      r := (v + (r/2)) / r;
	end_if;
  else // C -> temperature
    r := v * r;
  end_if;

END_FUNCTION

FUNCTION S_Weight2Kilogram VAR_INPUT v:DINT; p:^_VARIABLE; d:BOOL; END_VAR VAR_OUTPUT r:DINT; END_VAR

  r$udint := GetMulDiv(10000, p^.info.posdezpt);

  if(d = true) then // weight -> kg
    if(v < 0) then
      r := (v - (r/2)) / r;
	else
      r := (v + (r/2)) / r;
    end_if;
  else // kg -> weight
    r := v * r;
  end_if;

END_FUNCTION

FUNCTION S_Time2Second VAR_INPUT v:DINT; p:^_VARIABLE; d:BOOL; END_VAR VAR_OUTPUT r:DINT; END_VAR

  r$udint := GetMulDiv(1sec, p^.info.posdezpt);

  if(d = true) then
    if(v < 0) then
      r := (v - (r/2)) / r;
	else
      r := (v + (r/2)) / r;
    end_if;
  else
    r := v * r;
  end_if;

END_FUNCTION

FUNCTION S_Time2Minute VAR_INPUT v:DINT; p:^_VARIABLE; d:BOOL; END_VAR VAR_OUTPUT r:DINT; END_VAR

  if(d = true) then
    if(v < 0) then
      r := S_Time2Second((v-30)/60, p, true);
	else
      r := S_Time2Second((v+30)/60, p, true);
    end_if;
  else
    r := S_Time2Second(v*60, p, false);
  end_if;

END_FUNCTION

FUNCTION S_Time2Hour VAR_INPUT v:DINT; p:^_VARIABLE; d:BOOL; END_VAR VAR_OUTPUT r:DINT; END_VAR

  if(d = true) then
    if(v < 0) then
      r := S_Time2Minute((v-30)/60, p, true);
	else
      r := S_Time2Minute((v+30)/60, p, true);
    end_if;
  else
    r := S_Time2Minute(v*60, p, false);
  end_if;

END_FUNCTION

FUNCTION S_Pressure2Bar VAR_INPUT v:DINT; p:^_VARIABLE; d:BOOL; END_VAR VAR_OUTPUT r:DINT;END_VAR

  r$udint := GetMulDiv(1bar, p^.info.posdezpt);

  if(d = true) then
    if(v < 0) then
      r := (v - (r/2)) / r; // pressure -> bar
    else
      r := (v + (r/2)) / r; // pressure -> bar
	end_if;
  else
    r := v * r; // bar -> pressure
  end_if;

END_FUNCTION

FUNCTION S_Stroke2inch VAR_INPUT v:DINT; p:^_VARIABLE; d:BOOL; END_VAR VAR_OUTPUT r:DINT; END_VAR

  r$udint := GetMulDiv(1mm, p^.info.posdezpt) * 254;

  if(d = true) then // stroke -> inch
    if(v < 0) then
      r := ((v * 10) - (r / 2)) / r;
	else
      r := ((v * 10) + (r / 2)) / r;
    end_if;
  else // inch -> stroke
    r := ((v * r) + 5) / 10;
  end_if;

END_FUNCTION

FUNCTION S_Pressure2Psi VAR_INPUT v:DINT; p:^_VARIABLE; d:BOOL; END_VAR VAR_OUTPUT r:DINT; END_VAR
  var
    rv : real;
  end_var

  rv := R_Pressure2Psi(v, p, d);
  r  := to_dint(MyRealCalc(rv, p^.info.posdezpt, d));

END_FUNCTION

FUNCTION S_Weight2Pound VAR_INPUT v:DINT; p:^_VARIABLE; d:BOOL; END_VAR VAR_OUTPUT r:DINT; END_VAR
  var
    rv : real;
  end_var

  rv := R_Weight2Pound(v, p, d);
  r  := to_dint(MyRealCalc(rv, p^.info.posdezpt, d));

END_FUNCTION

FUNCTION S_Temp2Fahrenheit VAR_INPUT v:DINT; p:^_VARIABLE; d:BOOL; END_VAR VAR_OUTPUT r:DINT; END_VAR
  // lasal grundeinheit : 10E-1 Grad C
  // [C] = ([F]-32)*5/9

  if(d = true) then
    if(v < 0) then
      r := (((v * 9) - 2) / 5) + 320;
	else
      r := (((v * 9) + 2) / 5) + 320;
    end_if;
    if(p^.info.posdezpt = 0) then
	  if(r < 0) then
        r := (r - 5) / 10;
	  else
        r := (r + 5) / 10;
      end_if;
    end_if;
  else
    if(p^.info.posdezpt = 0) then
      r := (v - 32) * 10;
    else
      r := v - 320;
    end_if;

	if(r < 0) then
      r := ((r * 5) - 4) / 9;
	else
      r := ((r * 5) + 4) / 9;
    end_if;
  end_if;

END_FUNCTION

FUNCTION S_Force2KN VAR_INPUT v:DINT; p:^_VARIABLE; d:BOOL; END_VAR VAR_OUTPUT r:DINT; END_VAR

  r$udint := GetMulDiv(1kn, p^.info.posdezpt);

  if(d = true) then
    if(v < 0) then
      r := (v - (r/2)) / r; // force -> KN
    else
      r := (v + (r/2)) / r; // force -> KN
    end_if;
  else
    r := v * r; // KN -> force
  end_if;

END_FUNCTION

//[#ENGLISH]
//function is called in case of an recalculation (formula) defined for a data-server
//pres ....... --> to value
//pv ......... --> to variable
//direction .. direction (TRUE Y=kX+d, FALSE X=(Y+d)/k)
//retcode .... return TRUE if kernel should do the calculation, on the other hand return FALSE
FUNCTION __CDECL VIRTUAL GLOBAL _Lse::IF_Recalculate
VAR_INPUT
	pres		: ^_RESULT;
	pv          : ^_VARIABLE;
	direction   : BOOL;
END_VAR
VAR_OUTPUT
    retcode : BOOL;
END_VAR
VAR
 #ifndef CUTOFF_USER
  no   : UDINT;
  ppp  : ^_POINTERPARA;
 #endif
END_VAR

  retcode := TRUE;

 #ifndef CUTOFF_USER
  if(GlobalBitState and GLOBAL_BIT_IFRECALCULATE) then
    no  := UserGlobal.no;
    ppp := UserGlobal.ptr;
    while no do
      no  -= 1;
      if(ppp^.para and GLOBAL_BIT_IFRECALCULATE) then
        if(ppp^.ptr$^_Global^.IF_Recalculate(pres, pv, direction) = FALSE) then
          no := 0;
          retcode := FALSE;
        end_if;
      end_if;
      ppp += sizeof(_POINTERPARA);
    end_while;
  end_if;
 #endif

  if(retcode = TRUE) then
    retcode := FALSE;
   #ifdef UC_REAL
    if(pres^.ftype = RES_REAL) then
      case(pv^.info.formula) of
         3 : pres^.value$REAL := R_Stroke2mm(pres^.value$REAL, pv, direction);
         4 : pres^.value$REAL := R_Stroke2inch(pres^.value$REAL, pv, direction);
         5 : pres^.value$REAL := R_Temp2Celsius(pres^.value$REAL, pv, direction);
         6 : pres^.value$REAL := R_Temp2Fahrenheit(pres^.value$REAL, pv, direction);
         7 : pres^.value$REAL := R_Weight2Kilogram(pres^.value$REAL, pv, direction);
         8 : pres^.value$REAL := R_Weight2Pound(pres^.value$REAL, pv, direction);
         9 : pres^.value$REAL := R_Pressure2Bar(pres^.value$REAL, pv, direction);
        10 : pres^.value$REAL := R_Pressure2Psi(pres^.value$REAL, pv, direction);
        11 : pres^.value$REAL := R_Time2Second(pres^.value$REAL, pv, direction);
        12 : pres^.value$REAL := R_Time2Minute(pres^.value$REAL, pv, direction);
        13 : pres^.value$REAL := R_Time2Hour(pres^.value$REAL, pv, direction);
        14 : pres^.value$REAL := R_Force2KN(pres^.value$REAL, pv, direction);
		else retcode := TRUE;
	  end_case;
	else
   #endif
      case(pv^.info.formula) of
         3 : pres^.value := S_Stroke2mm(pres^.value, pv, direction);
         4 : pres^.value := S_Stroke2inch(pres^.value, pv, direction);
         5 : pres^.value := S_Temp2Celsius(pres^.value, pv, direction);
         6 : pres^.value := S_Temp2Fahrenheit(pres^.value, pv, direction);
         7 : pres^.value := S_Weight2Kilogram(pres^.value, pv, direction);
         8 : pres^.value := S_Weight2Pound(pres^.value, pv, direction);
         9 : pres^.value := S_Pressure2Bar(pres^.value, pv, direction);
        10 : pres^.value := S_Pressure2Psi(pres^.value, pv, direction);
        11 : pres^.value := S_Time2Second(pres^.value, pv, direction);
        12 : pres^.value := S_Time2Minute(pres^.value, pv, direction);
        13 : pres^.value := S_Time2Hour(pres^.value, pv, direction);
        14 : pres^.value := S_Force2KN(pres^.value, pv, direction);
		else retcode := TRUE;
	  end_case;
   #ifdef UC_REAL
	end_if;
   #endif

  end_if;

END_FUNCTION

FUNCTION VIRTUAL GLOBAL _Lse::Lse::NewInst
VAR_INPUT
 pPara  : ^CmdStruct;
 pResult  : ^Results;
END_VAR
VAR_OUTPUT
 ret_code  : IprStates;
END_VAR

  ret_code:= READY;

  CASE pPara^.uiCmd OF

    0:  // download start
      DownloadState := 1;
      pResult^.aData[0]$UDINT := 16#46544F44; // DOTF-id
      pResult^.uiLng          := 6;

    1:  // download finished
      DownloadState := 2;
      pResult^.aData[0]$UDINT := 16#46544F44; // DOTF-id
      pResult^.uiLng          := 6;

  END_CASE;

END_FUNCTION

FUNCTION VIRTUAL GLOBAL _Lse::IF_STOP
VAR_OUTPUT
	retcode		: BOOL;
END_VAR
VAR
	no   : UDINT;
	ppp  : ^_POINTERPARA;
END_VAR

  retcode := true;
//  InsertCmd(CMD_NEWPICTURE, get_startpicture(), 0);

  no  := UserGlobal.no;
  ppp := UserGlobal.ptr;
  while no do
    no  -= 1;
    if(ppp^.ptr$^_Global^.IF_Stop() = false) then
      retcode := false;
    end_if;
    ppp += sizeof(_POINTERPARA);
  end_while;

  if(retcode = false) then
    do_start();
  end_if;

END_FUNCTION

FUNCTION __CDECL VIRTUAL GLOBAL _Lse::IF_Online
VAR_INPUT
	station		: UINT;
END_VAR
VAR
	no   : UDINT;
	ppp  : ^_POINTERPARA;
END_VAR

  no  := UserGlobal.no;
  ppp := UserGlobal.ptr;
  while no do
    ppp^.ptr$^_Global^.IF_Online(station);
    no  -= 1;
    ppp += sizeof(_POINTERPARA);
  end_while;

END_FUNCTION

FUNCTION __CDECL VIRTUAL GLOBAL _Lse::IF_TryToAccess
VAR_INPUT
	ptx		: ^void;
	state		: _ACCESSFAILED;
	found		: _FOUNDHID;
	preselect		: bool;
END_VAR
VAR_OUTPUT
	retcode		: bool;
END_VAR
VAR
	no   : UDINT;
	ppp  : ^_POINTERPARA;
END_VAR

  retcode := preselect;

  if(GlobalBitState and GLOBAL_BIT_IFTRYTOACCESS) then
    no      := UserGlobal.no;
    ppp     := UserGlobal.ptr;
    while no do
      no      -= 1;
      if(ppp^.para and GLOBAL_BIT_IFTRYTOACCESS) then
        retcode := ppp^.ptr$^_Global^.IF_TryToAccess(ptx, state, found, preselect);
        if(retcode <> preselect) then
          no := 0;
        end_if;
      end_if;
      ppp += sizeof(_POINTERPARA);
    end_while;
  end_if;

END_FUNCTION

FUNCTION __CDECL VIRTUAL GLOBAL _Lse::IF_CheckHeap
VAR_INPUT
	display		: bool;
END_VAR
VAR_OUTPUT
	retcode		: _DOIT;
END_VAR
VAR
	no   : UDINT;
	ppp  : ^_POINTERPARA;
END_VAR

  retcode    := _IDLE;

  no  := UserGlobal.no;
  ppp := UserGlobal.ptr;
  while no do
    retcode := ppp^.ptr$^_Global^.IF_CheckHeap(display);
    no  -= 1;
    ppp += sizeof(_POINTERPARA);
    if(retcode <> _IDLE) then
      no := 0;
    end_if;
  end_while;

END_FUNCTION

FUNCTION __CDECL VIRTUAL GLOBAL _Lse::IF_SwitchMultiStation
VAR_INPUT
	station		: UINT;
END_VAR
VAR
	no   : UDINT;
	ppp  : ^_POINTERPARA;
END_VAR

  no  := UserGlobal.no;
  ppp := UserGlobal.ptr;
  while no do
    ppp^.ptr$^_Global^.IF_SwitchMultiStation(station);
    no  -= 1;
    ppp += sizeof(_POINTERPARA);
  end_while;

END_FUNCTION

#pragma warning (disable : 73)
FUNCTION __CDECL VIRTUAL GLOBAL _Lse::DoCmdInterface
VAR_INPUT
	cmd		: _PIC_COMMAND;
	op1		: DINT;
	op2		: DINT;
	psl		: ^_STACK_LINE;
END_VAR
VAR_OUTPUT
	retcode	: BOOL;
END_VAR

  retcode := true;

END_FUNCTION
#pragma warning (default: 73)

FUNCTION __CDECL VIRTUAL GLOBAL _Lse::IF_ScreenSaverWillStart
VAR_OUTPUT
	retcode		: bool;
END_VAR
VAR
	no  : UDINT;
	ppp  : ^_POINTERPARA;
END_VAR

  retcode := true;

  no  := UserGlobal.no;
  ppp := UserGlobal.ptr;
  while no do
    retcode := ppp^.ptr$^_Global^.IF_ScreenSaverWillStart();
    no  -= 1;
    ppp += sizeof(_POINTERPARA);
    if(retcode = _FALSE) then
      no := 0;
    end_if;
  end_while;

END_FUNCTION

FUNCTION __CDECL VIRTUAL GLOBAL _Lse::IF_ScreenSaverWillEnd
VAR_INPUT
    pev : ^_EVENT;
END_VAR
VAR_OUTPUT
	retcode		: bool;
END_VAR
VAR
	no  : UDINT;
	ppp  : ^_POINTERPARA;
END_VAR

  retcode := true;

  no  := UserGlobal.no;
  ppp := UserGlobal.ptr;
  while no do
    retcode := ppp^.ptr$^_Global^.IF_ScreenSaverWillEnd(pev);
    no  -= 1;
    ppp += sizeof(_POINTERPARA);
    if(retcode = _FALSE) then
      no := 0;
    end_if;
  end_while;

END_FUNCTION

FUNCTION __CDECL VIRTUAL GLOBAL _Lse::IF_Beep
  VAR_INPUT
    whobeep 	: _WHOBEEP;
  END_VAR
  VAR
    no  : UDINT;
	  ppp  : ^_POINTERPARA;
  END_VAR

  no  := UserGlobal.no;
  ppp := UserGlobal.ptr;
  while no do
    ppp^.ptr$^_Global^.IF_Beep(whobeep);
    no  -= 1;
    ppp += sizeof(_POINTERPARA);
  end_while;

END_FUNCTION

FUNCTION __CDECL VIRTUAL GLOBAL _Lse::IF_IpcIni
  VAR_INPUT
    pini 	: ^_IPCINI;
  END_VAR
  VAR
    no  : UDINT;
    ppp  : ^_POINTERPARA;
  END_VAR

  no  := UserGlobal.no;
  ppp := UserGlobal.ptr;
  while no do
    ppp^.ptr$^_Global^.IF_IpcIni(pini);
    no  -= 1;
    ppp += sizeof(_POINTERPARA);
  end_while;

END_FUNCTION

#pragma warning (disable: 73)
//[#ENGLISH]
//diese funktion wandelt eine zahl (4 Byte) in einen string um.
//die darstellung im string erfolgt hexadezimal.
//bitweise darstellung von format:
//.... .... .... **** no of digits
//.... .... **** .... position decimalpoint
//.... ...* .... .... preceding zeros
//.... ..*. .... .... descendant zeros
//.... .*.. .... .... vorzeichen unmittelbar vor wert (-3 ansonsten -  3)
//.... *... .... .... anzahl der stellen automatisch ermitteln
FUNCTION VIRTUAL GLOBAL _Lse::Str_DToH
VAR_INPUT
  pt       : ^VOID;
  value    : DINT;
  format   : UINT;
  chr_size : UINT;
END_VAR

  Lse_DToH(pt, value, format, chr_size);

END_FUNCTION

//[#ENGLISH]
//diese funktion wandelt eine zahl (4 Byte) in einen string um.
//die darstellung im string erfolgt dezimal.
//bitweise darstellung von format:
//.... .... .... **** no of digits
//.... .... **** .... position decimalpoint
//.... ...* .... .... preceding zeros
//.... ..*. .... .... descendant zeros
//.... .*.. .... .... vorzeichen unmittelbar vor wert (-3 ansonsten -  3)
//.... *... .... .... anzahl der stellen automatisch ermitteln
FUNCTION VIRTUAL GLOBAL _Lse::Str_DToA
VAR_INPUT
  pt       : ^VOID;
  value    : DINT;
  format   : UINT;
  chr_size : UINT;
END_VAR

  Lse_DToA(pt, value, format, chr_size);

END_FUNCTION

//[#ENGLISH]
//diese funktion ermittelt die anzahl der zeichen in einem string.
//der string wird mittels parameter txt bekanntgegeben.
//der parameter chr_size gibt auskunft ueber die groesse eines zeichens. (ASCII oder UNI code)
FUNCTION VIRTUAL GLOBAL _Lse::Str_Len
VAR_INPUT
  txt       : ^VOID;
  chr_size : UINT;
END_VAR
VAR_OUTPUT
  retcode : UINT;
END_VAR

  retcode := Lse_StrLen(txt, chr_size);

END_FUNCTION

//[#ENGLISH]
// diese funktion kopiert den string pt2 nach pt1.
// die parameter size1 und size2 geben auskunft ueber die jeweilige zeichengroesse
// uni und ascii-code string duerfen gemischt werden
FUNCTION VIRTUAL GLOBAL _Lse::Str_Cpy
VAR_INPUT
  pt1   : ^VOID;
  size1 : UINT;
  pt2   : ^VOID;
  size2 : UINT;
END_VAR

  Lse_StrCpy(pt1, size1, pt2, size2);

END_FUNCTION

//[#ENGLISH]
// diese funktion kopiert den string pt2 an das ende von pt1.
// die parameter size1 und size2 geben auskunft ueber die jeweilige zeichengroesse
// uni und ascii-code string duerfen gemischt werden
FUNCTION VIRTUAL GLOBAL _Lse::Str_Cat
VAR_INPUT
  pt1   : ^VOID;
  size1 : UINT;
  pt2   : ^VOID;
  size2 : UINT;
END_VAR

  Lse_StrCat(pt1, size1, pt2, size2);

END_FUNCTION

//[#ENGLISH]
// diese funktion vergleicht den string pt2 mit string pt1.
// die parameter size1 und size2 geben auskunft ueber die jeweilige zeichengroesse
// uni und ascii-code string duerfen gemischt werden
// sind beide strings ident so wird 0 zurueckgeliefert, ansonsten <>0
FUNCTION VIRTUAL GLOBAL _Lse::Str_Cmp
VAR_INPUT
  pt1   : ^VOID;
  size1 : UINT;
  pt2   : ^VOID;
  size2 : UINT;
END_VAR
VAR_OUTPUT
  retcode : UINT;
END_VAR

  retcode := Lse_StrCmp(pt1, size1, pt2, size2);

END_FUNCTION

//[#ENGLISH]
//diese funktion berechnet die größe eines strings in byte,
//wobei jedoch die abschließende 0 nicht mitgerechnet wird.
FUNCTION VIRTUAL GLOBAL _Lse::Str_Size
VAR_INPUT
  pt1   : ^VOID;
  size1 : UINT;
END_VAR
VAR_OUTPUT
  retcode : UINT;
END_VAR

  retcode := Lse_StrSize(pt1, size1);

END_FUNCTION

//[#ENGLISH]
//diese funktion sucht nach dem zeichen c im string p und gibt dessen position
//zurück. ist das zeichen c nicht im string vorhanden, so wird der wert 16#FFFF (65535) zurückgegeben.
//nach 0 (stringende) kann nicht gesucht werden; verwenden sie hierfür die funktion Str_Len().
FUNCTION VIRTUAL GLOBAL _Lse::Str_Chr
VAR_INPUT
  pt1   : ^VOID;
  chr   : _UNI;
  size1 : UINT;
END_VAR
VAR_OUTPUT
  retcode : UINT;
END_VAR

  retcode := Lse_StrChr(pt1, chr, size1);

END_FUNCTION

//[#ENGLISH]
//im string pt1 werden alle kleinbuchstaben [a-z] auf großbuchstaben [A-Z] geändert.
//der parameter len gibt an, bis zu welcher position im string die zeichen geändert werden sollten.
//ist len gleich 0, so wird der gesamte string durchsucht.
FUNCTION VIRTUAL GLOBAL _Lse::Str_Up
VAR_INPUT
  pt1   : ^VOID;
  size1 : UINT;
  len   : UINT;
END_VAR

  Lse_StrUp(pt1, size1, len);

END_FUNCTION

FUNCTION VIRTUAL GLOBAL _Lse::Out_ParameterString
VAR_INPUT
  room : _ROOM;
  pt   : ^_CHAR;
  pv   : ^_MEM_VARLABEL;
  font : _FONT;
  att  : _ATTRIB;
  col  : _COLOR;
END_VAR

  Lse_OutParaString(#room, pt, pv, font, att, col);

END_FUNCTION

//[#DEUTSCH]
//Diese Funktion gibt einen Text, der mittels dem Parameter txt angegeben ist
//im definierten Bereich (pr) aus.
//
//Parameter :
//txt     ^_CHAR    Pointer auf einen text
//pr     ^_ROOM   Pointer auf den Bereich
//font  _FONT       Schriftart
//att    _ATTRIB    Attribute (z.B T_BOLD "fett")
//col   _COLOR     Farbe des Textes
//[#ENGLISH]
//Diese Funktion gibt einen Text, der mittels dem Parameter txt angegeben ist
//im definierten Bereich (pr) aus.
//
//Parameter :
//txt     ^_CHAR    Pointer auf einen text
//pr     ^_ROOM   Pointer auf den Bereich
//font  _FONT       Schriftart
//att    _ATTRIB    Attribute (z.B T_BOLD "fett")
//col   _COLOR     Farbe des Textes
FUNCTION VIRTUAL GLOBAL _Lse::Out_TextAlign
VAR_INPUT
  txt  : ^_CHAR;
  pr   : ^_ROOM;
  font : _FONT;
  att  : _ATTRIB;
  col  : _COLOR;
END_VAR

  Lse_OutTextAlign(txt, pr, font, att, col);

END_FUNCTION

FUNCTION VIRTUAL GLOBAL _Lse::Lib_FormatValue
VAR_INPUT
  txt   : ^_CHAR;
  value : _IVALUE;
  pi1   : ^_VARINFO;
  pf1   : ^_PICFORMAT;
END_VAR

  format_value(txt, value, pi1, pf1);

END_FUNCTION

FUNCTION VIRTUAL GLOBAL _Lse::Lib_FormatTime
VAR_INPUT
  txt    : ^_CHAR;
  pt1    : ^_TIME;
  format : UINT;
END_VAR

  format_time(txt, pt1, format);

END_FUNCTION

FUNCTION VIRTUAL GLOBAL _Lse::Lib_FormatDate
VAR_INPUT
  txt    : ^_CHAR;
  pt1    : ^_DATE;
  format : UINT;
END_VAR

  format_date(txt, pt1, format);

END_FUNCTION

FUNCTION VIRTUAL GLOBAL _Lse::BMP_Draw
VAR_INPUT
  x1   : _KOORD;
  y1   : _KOORD;
  dpne : ^_ASCII;
END_VAR
VAR_OUTPUT
  retcode : BOOL;
END_VAR

 #ifdef UC_IPC
  retcode := flash_bmp(x1, y1, dpne);
 #else
  retcode := FALSE;
 #endif

END_FUNCTION

FUNCTION VIRTUAL GLOBAL _Lse::BMP_Save
VAR_INPUT
  dpne : ^_ASCII;
  x1   : _KOORD;
  y1   : _KOORD;
  x2   : _KOORD;
  y2   : _KOORD;
END_VAR
VAR_OUTPUT
  retcode : BOOL;
END_VAR

 #ifdef UC_IPC
  retcode := save_bmp(dpne, x1, y1, x2, y2, FALSE);
 #else
  retcode := FALSE;
 #endif

END_FUNCTION

FUNCTION VIRTUAL GLOBAL _Lse::Fnt_Size
VAR_INPUT
  fnt : _FONT;
  x   : ^UINT;
  y   : ^UINT;
END_VAR

  font_size(fnt, x, y);

END_FUNCTION

FUNCTION VIRTUAL GLOBAL _Lse::Fnt_Set
VAR_INPUT
  fnt : _FONT;
END_VAR
VAR_OUTPUT
  retcode : BOOL;
END_VAR

  font_set(fnt);
  retcode := TRUE;

END_FUNCTION

FUNCTION VIRTUAL GLOBAL _Lse::Fnt_Seek
VAR_INPUT
  name : ^_ASCII;
END_VAR
VAR_OUTPUT
  retcode : UINT;
END_VAR

  retcode := font_seek(name);

END_FUNCTION

FUNCTION VIRTUAL GLOBAL _Lse::VarLst_GetVarInfo
VAR_INPUT
  pvi  : ^_VARINFO;
  no   : UDINT;
END_VAR
VAR_OUTPUT
  retcode : BOOL;
END_VAR

  retcode := VarList_GetVarInfo(pvi, no);

END_FUNCTION

//[#ENGLISH]
//this function gets the whole information about a variable
//pvi ... --> to structure where information will be stored
//no .... number of variable
//if required variable is inaccessible, method returns FALSE on the other hand TRUE
FUNCTION VIRTUAL GLOBAL _Lse::VarLst_GetSingleVariable
VAR_INPUT
  pv : ^_VARIABLE;
  no : UDINT;
END_VAR
VAR_OUTPUT
  retcode : BOOL;
END_VAR

  retcode := VarList_GetSingleVariable(pv, no);

END_FUNCTION

//[#ENGLISH]
//this function gets the whole information about a variable
//pvi ... --> to structure where information will be stored
//pvl ... --> to information where variable is adressed
//if required variable is inaccessible, method returns FALSE on the other hand TRUE
FUNCTION VIRTUAL GLOBAL _Lse::VarLst_GetVariable
VAR_INPUT
  pv      : ^_VARIABLE;
  pvl     : ^_VARLABEL;
END_VAR
VAR_OUTPUT
  retcode : BOOL;
END_VAR

  retcode := VarList_GetVariable(pv, pvl);

END_FUNCTION

//[#ENGLISH]
//use this method to get data which are defined by a _VARLABEL
//pr ........ --> to structure where required data will be stored
//pv ........ --> to structure where whole information about variable will be stored
//pvl ....... --> to _VARLABEL which adresses your variable, maybe it could be a constant, date, time etc.
//wait4plc .. TRUE means i want to wait till data are ready
//if required variable is inaccessible, method returns FALSE on the other hand TRUE
FUNCTION VIRTUAL GLOBAL _Lse::VarLst_GetSystemData
VAR_INPUT
  pr       : ^_RESULT;
  pv       : ^_VARIABLE;
  pvl      : ^_VARLABEL;
  wait4plc : BOOL;
END_VAR
VAR_OUTPUT
  retcode : BOOL;
END_VAR

  retcode := VarList_GetSystemData(pr, pv, pvl, wait4plc);

END_FUNCTION

//[#ENGLISH]
//this method returns the size of a variable which is defined by parameter pv
//pv ... --> to structure which keeps information about variable
//method returns no of bytes. example: sizeof(DINT) or sizeof(USINT)
FUNCTION VIRTUAL GLOBAL _Lse::VarLst_GetVariableSize
VAR_INPUT
  pv      : ^_VARINFO;
END_VAR
VAR_OUTPUT
  retcode : UINT;
END_VAR

  retcode := VarList_GetVariableSize(pv);

END_FUNCTION

//[#ENGLISH]
//use this method to set data which are defined by a _VARLABEL
//pr ............. --> to structure who keeps data to store
//pv ............. --> to structure where whole information about variable will be stored
//pvl ............ --> to _VARLABEL which adresses your variable
//saveimmediate .. TRUE means i want to store data immediately
//if datas are stored, method returns TRUE on the other hand FALSE
FUNCTION VIRTUAL GLOBAL _Lse::VarLst_SetSystemData
VAR_INPUT
  pr            : ^_RESULT;
  pv            : ^_VARIABLE;
  pvl           : ^_VARLABEL;
  saveimmediate : BOOL;
END_VAR
VAR_OUTPUT
  retcode : BOOL;
END_VAR

  retcode := VarList_SetSystemData(pr, pv, pvl, saveimmediate);

END_FUNCTION

//[#ENGLISH]
//use this method to get data from a server which is adressed by servernumber
//note: function works just in case of numeric server (no time, date, string...)
//pn ......... servernumber
//pval ....... --> to memorylocation where serverdata should be stored
//wait4plc ... TRUE means i want to wait till data are ready
//if server-data is valid, method returns TRUE on the other hand FALSE
FUNCTION VIRTUAL GLOBAL _Lse::VarLst_GetValueByNo
VAR_INPUT
  no       : UDINT;
  pval     : ^_IVALUE;
  wait4plc :  BOOL;
END_VAR
VAR_OUTPUT
  retcode : BOOL;
END_VAR

  retcode := VarList_GetValueByNo(no, pval, wait4plc);

END_FUNCTION

//[#ENGLISH]
//use this method to get data which are defined by a _VARLABEL
//note: function works just in case of numeric server (no time, date, string...)
//pvl ........ --> to _VARLABEL which adresses your server
//pd ......... --> to memorylocation where serverdata should be stored
//wait4plc ... TRUE means i want to wait till data are ready
//if datas are stored, method returns TRUE on the other hand FALSE
FUNCTION VIRTUAL GLOBAL _Lse::VarLst_GetValue
VAR_INPUT
  pvl      : ^_VARLABEL;
  pd       : ^_IVALUE;
  wait4plc : BOOL;
END_VAR
VAR_OUTPUT
  retcode : BOOL;
END_VAR

  retcode := VarList_GetValue(pvl, pd, wait4plc);

END_FUNCTION

FUNCTION VIRTUAL GLOBAL _Lse::VarLst_SetValueByNo
VAR_INPUT
  no    : UDINT;
  value : DINT;
END_VAR
VAR_OUTPUT
  retcode : BOOL;
END_VAR

  retcode := VarList_SetValueByNo(no, value);

END_FUNCTION

FUNCTION VIRTUAL GLOBAL _Lse::VarLst_GetCompleteNoDigits
VAR_INPUT
  pvi : ^_VARINFO;
END_VAR
VAR_OUTPUT
  retcode : UINT;
END_VAR

  retcode := VarList_GetCompleteNoDigits(pvi);

END_FUNCTION

FUNCTION VIRTUAL GLOBAL _Lse::VarLst_GetLabel
VAR_INPUT
  pd  : ^_ASCII;
  no  : UDINT;
END_VAR
VAR_OUTPUT
  retcode : BOOL;
END_VAR
VAR
  dummy : _UBYTE;
END_VAR
  retcode := VarList_GetLabel(pd, #dummy, no);

END_FUNCTION

FUNCTION VIRTUAL GLOBAL _Lse::VarLst_GetVarNo
VAR_INPUT
  plabel : ^_ASCII;
END_VAR
VAR_OUTPUT
  retcode : UDINT;
END_VAR

  retcode := VarList_GetVarNo(plabel);

END_FUNCTION

FUNCTION VIRTUAL GLOBAL _Lse::VarLst_GetTool
VAR_INPUT
  parameter : UDINT;
END_VAR
VAR_OUTPUT
  retcode : BOOL;
END_VAR

  retcode := VarList_GetParameter(parameter, 0);

END_FUNCTION

FUNCTION VIRTUAL GLOBAL _Lse::VarLst_GetProt
VAR_INPUT
  parameter : UDINT;
END_VAR
VAR_OUTPUT
  retcode : BOOL;
END_VAR

  retcode := VarList_GetParameter(parameter, 1);

END_FUNCTION

FUNCTION VIRTUAL GLOBAL _Lse::VarLst_GetPde
VAR_INPUT
  parameter : UDINT;
END_VAR
VAR_OUTPUT
  retcode : BOOL;
END_VAR

  retcode := VarList_GetParameter(parameter, 2);

END_FUNCTION

FUNCTION VIRTUAL GLOBAL _Lse::VarLst_GetZero
VAR_INPUT
  info : UINT;
END_VAR
VAR_OUTPUT
  retcode : BOOL;
END_VAR

  retcode := VarList_VOWPRUIC(info, 7);

END_FUNCTION

FUNCTION VIRTUAL GLOBAL _Lse::VarLst_GetRefr
VAR_INPUT
  info : UINT;
END_VAR
VAR_OUTPUT
  retcode : BOOL;
END_VAR

  retcode := VarList_VOWPRUIC(info, 3);

END_FUNCTION

FUNCTION VIRTUAL GLOBAL _Lse::VarLst_GetUser
VAR_INPUT
  info : UINT;
END_VAR
VAR_OUTPUT
  retcode : BOOL;
END_VAR

  retcode := VarList_VOWPRUIC(info, 2);

END_FUNCTION

FUNCTION VIRTUAL GLOBAL _Lse::VarLst_GetInvert
VAR_INPUT
  info : UINT;
END_VAR
VAR_OUTPUT
  retcode : BOOL;
END_VAR

  retcode := VarList_VOWPRUIC(info, 1);

END_FUNCTION

FUNCTION VIRTUAL GLOBAL _Lse::VarLst_GetText
VAR_INPUT
  no : UINT;
END_VAR
VAR_OUTPUT
  retcode : ^_CHAR;
END_VAR

  retcode := VarList_GetText(no);

END_FUNCTION

FUNCTION VIRTUAL GLOBAL _Lse::VarLst_GetDigits
VAR_INPUT
  pvi : ^_VARINFO;
END_VAR
VAR_OUTPUT
  retcode : UINT;
END_VAR

  retcode := VarList_GetDigits(pvi);

END_FUNCTION

FUNCTION VIRTUAL GLOBAL _Lse::VarLst_GetSign
VAR_INPUT
  pvi : ^_VARINFO;
END_VAR
VAR_OUTPUT
  retcode : BOOL;
END_VAR

  retcode := VarList_GetSign(pvi);

END_FUNCTION

FUNCTION VIRTUAL GLOBAL _Lse::VarLst_GetDezPoint
VAR_INPUT
  pvi : ^_VARINFO;
END_VAR
VAR_OUTPUT
  retcode : DINT;
END_VAR

  retcode := VarList_GetDezPoint(pvi);

END_FUNCTION

FUNCTION VIRTUAL GLOBAL _Lse::VarLst_GetNo
VAR_OUTPUT
  retcode : UDINT;
END_VAR

  retcode := VarList_GetNo();

END_FUNCTION

FUNCTION VIRTUAL GLOBAL _Lse::VarLst_GetUnitInfo
VAR_INPUT
  no : UINT;
END_VAR
VAR_OUTPUT
  retcode : ^_UNIT;
END_VAR

  retcode := VarList_GetUnitInfo(no);

END_FUNCTION

FUNCTION VIRTUAL GLOBAL _Lse::VarLst_GetUnitNo
VAR_INPUT
	punit		: ^_ASCII;
END_VAR
VAR_OUTPUT
	retcode		: UINT;
END_VAR

  retcode := VarList_GetUnitNo(punit);

END_FUNCTION

FUNCTION VIRTUAL GLOBAL _Lse::TxtLst_GetText
VAR_INPUT
  list   : _ANYLST;
  txtno  : UDINT;
END_VAR
VAR_OUTPUT
 retcode : ^_CHAR;
END_VAR
  retcode := textpuffer_getText(list, txtno);
END_FUNCTION

FUNCTION VIRTUAL GLOBAL _Lse::TxtLst_GetSize
VAR_INPUT
  list   : _ANYLST;
END_VAR
VAR_OUTPUT
 retcode : DINT;
END_VAR
  retcode := textpuffer_getSize(list);
END_FUNCTION

FUNCTION VIRTUAL GLOBAL _Lse::TxtLst_GetPtr
VAR_INPUT
  list   : _ANYLST;
END_VAR
VAR_OUTPUT
  retcode : ^_CHAR;
END_VAR
  retcode := textpuffer_getPtr(list);
END_FUNCTION

FUNCTION VIRTUAL GLOBAL _Lse::TxtLst_GetNo
VAR_INPUT
  list   : _ANYLST;
END_VAR
VAR_OUTPUT
  retcode : UDINT;
END_VAR
  retcode := textpuffer_getNo(list);
END_FUNCTION

//[#DEUTSCH]
//Diese Funktion liefert den Error-Status eines bereits geöffneten Handle zurück.
//Nach dem Aufruf von Lse_File_Close() kann diese Funktion nicht mehr verwendet
//werden.
//
//Rückgabewert:
//	TRUE     es ist bereits ein Fehler aufgetreten
//	FALSE 	 bis zu diesem Zeitpunkt kein Fehler aufgetreten
//Parameter:
//	handle: 	--> auf das eigentliche Handle
//[#ENGLISH]
//With this function you will get the error state of an already opened handle
//You can't use this function after calling the function  LSE_File_Close()
//
//returned value:
//	TRUE     it already exists an error
//	FALSE 	 	no error up to now
//Parameter:
//	handle: 	--> to handle
FUNCTION VIRTUAL GLOBAL  _Lse::File_GetError
VAR_INPUT
  filep   : ^_LSEFILE;
END_VAR
VAR_OUTPUT
  retcode : BOOL;
END_VAR

  retcode := Lse_File_GetError(filep);

END_FUNCTION

//[#ENGLISH]
//With this function you can set a file to an error. It will be necessary
// if you have to read a lot of bytes of the file,, but you haven't enough memory
//
//Parameter:
//	handle: 	--> to handle
//  ferr : 		error state
FUNCTION VIRTUAL GLOBAL  _Lse::File_SetError
VAR_INPUT
  filep : ^_LSEFILE;
  ferr  : _FILE_ERROR;
END_VAR

  Lse_File_SetError(filep, ferr);

END_FUNCTION

//[#ENGLISH]
//This function open a file with the defined parameter dpne. If you open a file with
//function you have to close the file with Lse_File_Close().
//
//returned value:
//	TRUE 		if file could be opened
//	FALSE 		error
//Parameter:
//	handle: 	--> to handle
//	state: File for reading (LOAD), writing(SAVE) or reading and writing (LOADSAVE) open
//	dpne: drive, path, name and extension of the file
//example:
//	handle : _FILE;
//	Lse_File_Open(#handle, LOAD, "C:\\TEST.TXT"); // read only
//	Lse_File_Open(#handle, SAVE, "C:\\TEST.TXT"); // write only
FUNCTION VIRTUAL GLOBAL  _Lse::File_Open
VAR_INPUT
  filep : ^_LSEFILE;
  state : _FILE_STATE;
  dpne  :  ^_ASCII;
END_VAR
VAR_OUTPUT
  retcode : BOOL;
END_VAR

  retcode := Lse_File_Open(filep, state, dpne);

END_FUNCTION

//[#ENGLISH]
// This function closes an already opened file (with Lse_File_Open() )
// the parameter is a pointer to the handle
//
//returned value:
//	TRUE
//	FALSE 	during  work with this handle an error occurred
//Parameter:
//	handle: 	--> to Handle
//
//example:
//	handle : _FILE;
//	Lse_File_Open(#handle, LOAD, "C:\\TEST.TXT"); // open File
//	Lse_File_Close(#handle); // close File
FUNCTION VIRTUAL GLOBAL  _Lse::File_Close
VAR_INPUT
  filep : ^_LSEFILE;
END_VAR
VAR_OUTPUT
  retcode : BOOL;
END_VAR

  retcode := Lse_File_Close(filep);

END_FUNCTION

//[#ENGLISH]
//This function delete a file with the defined parameter dpne.
//The file must be closed.
//
//returned value:
//	TRUE 		if file could be deleted
//	FALSE 		error
//Parameter:
//	handle: 	--> to handle
//	dpne: drive, path, name and extension of the file
//example:
//	handle : _FILE;
//	Lse_File_Remove(#handle, "C:\\TEST.TXT");
FUNCTION VIRTUAL GLOBAL _Lse::File_Remove
VAR_INPUT
	filep		: ^_LSEFILE;
	dpne		: ^_ASCII;
END_VAR
VAR_OUTPUT
	retcode		: BOOL;
END_VAR

  retcode := Lse_File_Remove(filep, dpne);

END_FUNCTION

//[#ENGLISH]
//With this function you will get the actual read or write pointer in the opened file
//
//returned value:
//	position of the actual read or write pointer
//Parameter:
//	handle: 	--> to Handle
FUNCTION VIRTUAL GLOBAL  _Lse::File_Tell
VAR_INPUT
  filep  : ^_LSEFILE;
END_VAR
VAR_OUTPUT
  retcode : _DWORD;
END_VAR

  retcode := Lse_File_Tell(filep);

END_FUNCTION

//[#ENGLISH]
//With this function you set the read or write pointer in the opened file
//on a defined position
//
//returned value:
//	TRUE	the new position of the pointer is ok
//	FALSE 	during moving of the pointer an error occurred
//Parameter:
//	handle: 	--> to Handle
//  offs :		new position of the filepointer
//  fromwhere :	fromwhere should the new position computed
//				SEEK_SET	from the startposition of the file
//				SEEK_CUR	offs is the new absolut position
//				SEEK_END	position is the last entry of the file
FUNCTION VIRTUAL GLOBAL  _Lse::File_Seek
VAR_INPUT
  filep     : ^_LSEFILE;
  offs      : _DWORD;
  fromwhere : _UWORD;
END_VAR
VAR_OUTPUT
  retcode : BOOL;
END_VAR

  retcode := Lse_File_Seek(filep, offs, fromwhere);

END_FUNCTION

//[#ENGLISH]
//With this function you will get the actual size of the file (bytes)
//
//returned value:
//	the actual size of the file in byte
//Parameter:
//	handle: 	--> to Handle
FUNCTION VIRTUAL GLOBAL  _Lse::File_Length
VAR_INPUT
  filep : ^_LSEFILE;
END_VAR
VAR_OUTPUT
 retcode : _DWORD;
END_VAR

  retcode := Lse_File_Length(filep);

END_FUNCTION

//[#ENGLISH]
//This function reads a defined size of bytes of an already opened file(handle)
//The bytes are saved to the adress of the paramter dst. An error processing is
//in integrated in the handle.It isn't necessary to check the returned value
//every time.
//It is important, that the file is opened for writing
//
//returned value:
//	TRUE 	success
//	FALSE 	error, you can't use the data on dst
//Parameter:
//	handle: 	--> to Handle
//	dst: 	--> to data area
//  size: size of the reading bytes
//example:
//	handle : _FILE;
//	word : INT;
//	retcode : BOOL;
//
//	Lse_File_Open(#handle, LOAD, "C:\\TEST.TXT"); // open File
//	Lse_File_Read(#handle, #word, sizeof(INT)); // read 2 Byte
//	Lse_File_Read(#handle, #word, sizeof(INT)); // read the next 2 Byte
//	retcode = Lse_File_Close(#handle); // close File including check success
FUNCTION VIRTUAL GLOBAL  _Lse::File_Read
VAR_INPUT
  filep : ^_LSEFILE;
  dest  :  pVoid;
  size  :  _UDWORD;
END_VAR
VAR_OUTPUT
  retcode : BOOL;
END_VAR

  retcode := Lse_File_Read(filep, dest, size);

END_FUNCTION

//[#ENGLISH]
//This function writes a defined size of bytes in an already opened file (handle)
//An error processing is in integrated in the handle.
//It isn't necessary to check the returned value every time
//It is important, that the file is opened for writing
//
//returned value:
//	TRUE 	success
//	FALSE 	error, data couldn't write in the file (handle)
//Parameter:
//	handle: 	--> to Handle
//	src: 	--> to data area
//	size: size of data to write
//example:
//	handle _FILE;
//	word INT;
//	retcode BOOL;
//
//	Lse_File_Open(#handle, SAVE, "C:\\TEST.TXT"); // open File
//	Lse_File_Write(#handle, "aa", sizeof(INT)); // write 2 Byte
//	Lse_File_Write(#handle, "bb", sizeof(INT)); // write the next 2 Byte
//	retcode = Lse_File_Close(#handle); // close File including check success
FUNCTION VIRTUAL GLOBAL  _Lse::File_Write
VAR_INPUT
  filep : ^_LSEFILE;
  dest  : pVoid;
  size  : _UDWORD;
END_VAR
VAR_OUTPUT
  retcode : BOOL;
END_VAR

  retcode := Lse_File_Write(filep, dest, size);

END_FUNCTION

//[#ENGLISH]
//This function is a further development of the read function
//It is used for reading one line of a TXT-file. This line will be saved in the adress
//of dst. This function searchs for CR and LF and so you have to define a maximum
//size of bytes for reading one line. Without the definition of maxsize you can get
//an system error
//
//returned value:
//	TRUE   success
//	FALSE 	error, you can't use the data on dst
//Parameter:
//	handle: 	--> to Handle
//	dst: 	--> to data area
//maxsize: maximum size of reading bytes
//exampple:
//	handle : _FILE ;
//	line : ARRAY[0..99] of _ASCII;
//	retcode : ;
//
//	Lse_File_Open(&handle, LOAD, "C:\\TEST.TXT"); // open file
//	Lse_File_Read(&handle, line, 100); // read first line
//	retcode = Lse_File_Close(&handle); // close file including check success
FUNCTION VIRTUAL GLOBAL  _Lse::File_Read_CRLF
VAR_INPUT
  filep : ^_LSEFILE;
  dest  : pVoid;
  maxsize : _UWORD;
END_VAR
VAR_OUTPUT
  retcode : BOOL;
END_VAR

  retcode := Lse_File_Read_CRLF(filep, dest$^char, maxsize);

END_FUNCTION

FUNCTION VIRTUAL GLOBAL _Lse::SCROLL_GetLinePosition
VAR_INPUT
  pt1 : ^_SCROLL;
  y   : UINT;
  pr  :^_ROOM;
END_VAR

  GetLinePosition_SCROLL(pt1, y, pr);

END_FUNCTION

FUNCTION VIRTUAL GLOBAL _Lse::SCROLL_OutLine
VAR_INPUT
  pt1   : ^_SCROLL;
  y     : UINT;
  no    : UINT;
  beam  : BOOL;
END_VAR

  OutLine_SCROLL(pt1, y, no, beam, TRUE);

END_FUNCTION

FUNCTION VIRTUAL GLOBAL _Lse::SCROLL_Beam
VAR_INPUT
  pt1   : ^_SCROLL;
  y     : UINT;
  no    : UINT;
  state : BOOL;
END_VAR

  Beam_SCROLL(pt1, y, no, state);

END_FUNCTION

FUNCTION VIRTUAL GLOBAL _Lse::SCROLL_ActBeam
VAR_INPUT
  pt1   : ^_SCROLL;
  state : BOOL;
END_VAR

  ActBeam_SCROLL(pt1, state);

END_FUNCTION

FUNCTION VIRTUAL GLOBAL _Lse::SCROLL_Draw
VAR_INPUT
  pt1  : ^_SCROLL;
  beam : BOOL;
END_VAR

  Draw_SCROLL(pt1, beam);

END_FUNCTION

FUNCTION VIRTUAL GLOBAL _Lse::SCROLL_Start
VAR_INPUT
  pt1 : ^_SCROLL;
END_VAR

  Start_SCROLL(pt1, TRUE);

END_FUNCTION

FUNCTION VIRTUAL GLOBAL _Lse::SCROLL_Ready
VAR_INPUT
  pt1  : ^_SCROLL;
  beam : BOOL;
END_VAR

  Ready_SCROLL(pt1, beam);

END_FUNCTION

FUNCTION VIRTUAL GLOBAL _Lse::SCROLL_Run
VAR_INPUT
  pt1    : ^_SCROLL;
  pevent : ^_EVENT;
END_VAR

  Run_SCROLL(pt1, pevent);

END_FUNCTION

FUNCTION VIRTUAL GLOBAL _Lse::SCROLL_End
VAR_INPUT
  pt1 : ^_SCROLL;
END_VAR

  End_SCROLL(pt1);

END_FUNCTION

FUNCTION VIRTUAL GLOBAL _Lse::SCROLL_OutPage
VAR_INPUT
  pt1 : ^_SCROLL;
END_VAR

  OutPage_SCROLL(pt1);

END_FUNCTION

FUNCTION VIRTUAL GLOBAL _Lse::SCROLL_ScrollUp
VAR_INPUT
  pt1 : ^_SCROLL;
END_VAR

  ScrollUp_SCROLL(pt1);

END_FUNCTION

FUNCTION VIRTUAL GLOBAL _Lse::SCROLL_ScrollDown
VAR_INPUT
  pt1 : ^_SCROLL;
END_VAR

  ScrollDown_SCROLL(pt1);

END_FUNCTION

FUNCTION VIRTUAL GLOBAL _Lse::SCROLL_GetPosition
VAR_INPUT
  pt1 : ^_SCROLL;
END_VAR
VAR_OUTPUT
  retcode : UINT;
END_VAR

  retcode := GetPosition_SCROLL(pt1);

END_FUNCTION

FUNCTION VIRTUAL GLOBAL _Lse::SCROLL_level_draw
VAR_INPUT
  pt1   : ^_LEVEL;
  horiz : BOOL;
END_VAR

  level_draw(pt1, horiz, TRUE);

END_FUNCTION

FUNCTION VIRTUAL GLOBAL _Lse::SCROLL_level_run
VAR_INPUT
  pt1   : ^_LEVEL;
  no    : DINT;
  pos   : DINT;
  horiz : BOOL;
END_VAR

  level_run(pt1, no, pos, horiz);

END_FUNCTION

FUNCTION __CDECL VIRTUAL GLOBAL _Lse::IF_SoftReset

  DownloadState := 2;

END_FUNCTION

FUNCTION __CDECL VIRTUAL GLOBAL _Lse::IF_UserStation
	VAR_INPUT
		station 	: UINT;
		pcd 	: ^_COMDEF;
		pobserve 	: ^BOOL;
	END_VAR
	VAR_OUTPUT
		retcode 	: BOOL;
	END_VAR
  VAR
	  no   : UDINT;
    ppp  : ^_POINTERPARA;
  END_VAR

  retcode    := true;
  no  := UserGlobal.no;
  ppp := UserGlobal.ptr;
  while no do
    no  -= 1;
    if(ppp^.ptr$^_Global^.IF_UserStation(station, pcd, pobserve) = false) then
      retcode := false;
    end_if;
    ppp += sizeof(_POINTERPARA);
  end_while;

END_FUNCTION

FUNCTION __CDECL VIRTUAL GLOBAL _Lse::IF_CantWriteNoAccess
	VAR_INPUT
		pres 	: ^_RESULT;
		pvl 	: ^_VARLABEL;
	END_VAR
	VAR_OUTPUT
		retcode 	: BOOL;
	END_VAR
  VAR
	  no   : UDINT;
    ppp  : ^_POINTERPARA;
  END_VAR

  retcode := false;
  no  := UserGlobal.no;
  ppp := UserGlobal.ptr;
  while no do
    no  -= 1;
    if(ppp^.ptr$^_Global^.IF_CantWriteNoAccess(pres, pvl) = true) then
      retcode := true;
    end_if;
    ppp += sizeof(_POINTERPARA);
  end_while;

END_FUNCTION

FUNCTION VIRTUAL GLOBAL _Lse::ActivateBubbleHelp::Write
	VAR_INPUT
		input (EAX) 	: DINT;
	END_VAR
	VAR_OUTPUT
		result (EAX) 	: DINT;
	END_VAR

	ActivateBubbleHelp := input;
 	result := ActivateBubbleHelp;

  if(result <> 0) then
    InsertCmd(CMD_KILLEDITOR, 0, 0);
  end_if;

END_FUNCTION

FUNCTION __CDECL GLOBAL Thread2_AddCmd
  VAR_INPUT
    pcmd : ^_Thread2CmdLine;
  END_VAR
  VAR_OUTPUT
    retcode : bool;
  END_VAR

  retcode := false;

  if(pcmd^.cmd <> T2_NONE) then
    if(MailBox2Handle <> NIL) then
      if(OS_MT_PutCond(MailBox2Handle, pcmd) = 1) then
        retcode := true;
      end_if;
    end_if;
  end_if;

END_FUNCTION

FUNCTION __CDECL GLOBAL _Lse::Thread2
	VAR_INPUT
		pthis 	: ^void;
	END_VAR
  VAR
  	t2cmdline : _Thread2CmdLine;
  END_VAR

  this := pthis$^_Lse;

  while(1) do
    if(OS_MT_GET(MailBox2Handle, #t2cmdline) = MTERROR_NONE) then // wait for cmd in mailbox
      RTK_Thread2(#t2cmdline);
    end_if;
    OS_MT_DELAY(1);
  end_while;

END_FUNCTION
